  MoveL 3384 to (-30.78, 36.52, 59.84) mm, rotated rx 180 ry 0 rz 180 deg; joints [-35.866, -23.626, 89.959, 60.959, 42.078, -53.201]
  MoveL 3385 to (-30.78, 36.52, 59.84) mm, rotated rx 180 ry 0 rz 180 deg; joints [-35.866, -23.626, 89.959, 60.959, 42.078, -53.201]
  Call Extruder(71.38542)
  MoveL 3386 to (-30.58, 36.45, 59.84) mm, rotated rx 180 ry 0 rz 180 deg; joints [-35.829, -23.61, 89.95, 60.933, 42.045, -53.186]
  MoveL 3387 to (-30.58, 36.45, 59.84) mm, rotated rx 180 ry 0 rz 180 deg; joints [-35.829, -23.61, 89.95, 60.933, 42.045, -53.186]
  Call Extruder(71.51620)
  MoveL 3388 to (-30.36, 36.38, 59.84) mm, rotated rx 180 ry 0 rz 180 deg; joints [-35.788, -23.591, 89.94, 60.905, 42.009, -53.17]
  MoveL 3389 to (-30.36, 36.38, 59.84) mm, rotated rx 180 ry 0 rz 180 deg; joints [-35.788, -23.591, 89.94, 60.905, 42.009, -53.17]
  Call Extruder(71.64643)
  MoveL 3390 to (-30.14, 36.32, 59.84) mm, rotated rx 180 ry 0 rz -180 deg; joints [-35.748, -23.573, 89.929, 60.877, 41.973, -53.153]
  MoveL 3391 to (-30.14, 36.32, 59.84) mm, rotated rx 180 ry 0 rz -180 deg; joints [-35.748, -23.573, 89.929, 60.877, 41.973, -53.153]
  Call Extruder(71.77608)
  MoveL 3392 to (-29.91, 36.25, 59.84) mm, rotated rx -180 ry 0 rz 180 deg; joints [-35.708, -23.555, 89.919, 60.848, 41.937, -53.137]
  MoveL 3393 to (-29.91, 36.25, 59.84) mm, rotated rx -180 ry 0 rz 180 deg; joints [-35.708, -23.555, 89.919, 60.848, 41.937, -53.137]
  Call Extruder(71.90518)
  MoveL 3394 to (-29.69, 36.18, 59.84) mm, rotated rx 180 ry 0 rz 180 deg; joints [-35.668, -23.536, 89.908, 60.82, 41.9, -53.121]
  MoveL 3395 to (-29.69, 36.18, 59.84) mm, rotated rx 180 ry 0 rz 180 deg; joints [-35.668, -23.536, 89.908, 60.82, 41.9, -53.121]
  Call Extruder(72.02025)
  MoveL 3396 to (-29.48, 36.14, 59.84) mm, rotated rx 180 ry 0 rz 180 deg; joints [-35.634, -23.518, 89.898, 60.797, 41.87, -53.108]
  MoveL 3397 to (-29.48, 36.14, 59.84) mm, rotated rx 180 ry 0 rz 180 deg; joints [-35.634, -23.518, 89.898, 60.797, 41.87, -53.108]
  Call Extruder(72.13487)
  MoveL 3398 to (-29.28, 36.09, 59.84) mm, rotated rx -180 ry 0 rz 180 deg; joints [-35.601, -23.5, 89.888, 60.775, 41.839, -53.096]
  MoveL 3399 to (-29.28, 36.09, 59.84) mm, rotated rx -180 ry 0 rz 180 deg; joints [-35.601, -23.5, 89.888, 60.775, 41.839, -53.096]
  Call Extruder(72.24904)
  MoveL 3400 to (-29.08, 36.05, 59.84) mm, rotated rx -180 ry 0 rz 180 deg; joints [-35.567, -23.482, 89.878, 60.752, 41.808, -53.084]
  MoveL 3401 to (-29.08, 36.05, 59.84) mm, rotated rx -180 ry 0 rz 180 deg; joints [-35.567, -23.482, 89.878, 60.752, 41.808, -53.084]
  Call Extruder(72.36276)
  MoveL 3402 to (-28.87, 36, 59.84) mm, rotated rx 180 ry 0 rz 180 deg; joints [-35.533, -23.463, 89.867, 60.73, 41.777, -53.072]
  MoveL 3403 to (-28.87, 36, 59.84) mm, rotated rx 180 ry 0 rz 180 deg; joints [-35.533, -23.463, 89.867, 60.73, 41.777, -53.072]
  Call Extruder(72.48818)
  MoveL 3404 to (-28.64, 35.96, 59.84) mm, rotated rx 180 ry 0 rz 180 deg; joints [-35.497, -23.443, 89.856, 60.705, 41.744, -53.059]
  MoveL 3405 to (-28.64, 35.96, 59.84) mm, rotated rx 180 ry 0 rz 180 deg; joints [-35.497, -23.443, 89.856, 60.705, 41.744, -53.059]
  Call Extruder(72.62516)
  MoveL 3406 to (-28.4, 35.91, 59.84) mm, rotated rx 180 ry 0 rz 180 deg; joints [-35.457, -23.42, 89.843, 60.679, 41.707, -53.045]
  MoveL 3407 to (-28.4, 35.91, 59.84) mm, rotated rx 180 ry 0 rz 180 deg; joints [-35.457, -23.42, 89.843, 60.679, 41.707, -53.045]
  Call Extruder(72.76152)
  MoveL 3408 to (-28.15, 35.86, 59.84) mm, rotated rx 180 ry 0 rz 180 deg; joints [-35.417, -23.398, 89.83, 60.652, 41.67, -53.03]
  MoveL 3409 to (-28.15, 35.86, 59.84) mm, rotated rx 180 ry 0 rz 180 deg; joints [-35.417, -23.398, 89.83, 60.652, 41.67, -53.03]
  Call Extruder(72.89728)
  MoveL 3410 to (-27.9, 35.81, 59.84) mm, rotated rx 180 ry 0 rz 180 deg; joints [-35.377, -23.375, 89.817, 60.626, 41.634, -53.016]
  MoveL 3411 to (-27.9, 35.81, 59.84) mm, rotated rx 180 ry 0 rz 180 deg; joints [-35.377, -23.375, 89.817, 60.626, 41.634, -53.016]
  Call Extruder(73.03243)
  MoveL 3412 to (-27.65, 35.76, 59.84) mm, rotated rx 180 ry 0 rz 180 deg; joints [-35.337, -23.352, 89.804, 60.599, 41.597, -53.002]
  MoveL 3413 to (-27.65, 35.76, 59.84) mm, rotated rx 180 ry 0 rz 180 deg; joints [-35.337, -23.352, 89.804, 60.599, 41.597, -53.002]
  Call Extruder(73.16696)
  MoveL 3414 to (-27.4, 35.71, 59.84) mm, rotated rx 180 ry 0 rz 180 deg; joints [-35.297, -23.33, 89.791, 60.573, 41.56, -52.988]
  MoveL 3415 to (-27.4, 35.71, 59.84) mm, rotated rx 180 ry 0 rz 180 deg; joints [-35.297, -23.33, 89.791, 60.573, 41.56, -52.988]
  Call Extruder(73.30089)
  MoveL 3416 to (-27.15, 35.66, 59.84) mm, rotated rx 180 ry 0 rz 180 deg; joints [-35.258, -23.307, 89.778, 60.547, 41.524, -52.974]
  MoveL 3417 to (-27.15, 35.66, 59.84) mm, rotated rx 180 ry 0 rz 180 deg; joints [-35.258, -23.307, 89.778, 60.547, 41.524, -52.974]
  Call Extruder(73.44875)
  MoveL 3418 to (-26.87, 35.61, 59.84) mm, rotated rx 180 ry 0 rz -180 deg; joints [-35.215, -23.281, 89.764, 60.518, 41.484, -52.959]
  MoveL 3419 to (-26.87, 35.61, 59.84) mm, rotated rx 180 ry 0 rz -180 deg; joints [-35.215, -23.281, 89.764, 60.518, 41.484, -52.959]
  Call Extruder(73.61048)
  MoveL 3420 to (-26.57, 35.56, 59.84) mm, rotated rx 180 ry 0 rz 180 deg; joints [-35.168, -23.252, 89.747, 60.488, 41.441, -52.944]
  MoveL 3421 to (-26.57, 35.56, 59.84) mm, rotated rx 180 ry 0 rz 180 deg; joints [-35.168, -23.252, 89.747, 60.488, 41.441, -52.944]
  Call Extruder(73.77149)
  MoveL 3422 to (-26.26, 35.51, 59.84) mm, rotated rx 180 ry 0 rz 180 deg; joints [-35.122, -23.223, 89.731, 60.458, 41.398, -52.929]
  MoveL 3423 to (-26.26, 35.51, 59.84) mm, rotated rx 180 ry 0 rz 180 deg; joints [-35.122, -23.223, 89.731, 60.458, 41.398, -52.929]
  Call Extruder(73.93177)
  MoveL 3424 to (-25.96, 35.47, 59.84) mm, rotated rx 180 ry 0 rz 180 deg; joints [-35.075, -23.194, 89.714, 60.428, 41.355, -52.913]
  MoveL 3425 to (-25.96, 35.47, 59.84) mm, rotated rx 180 ry 0 rz 180 deg; joints [-35.075, -23.194, 89.714, 60.428, 41.355, -52.913]
  Call Extruder(74.09132)
  MoveL 3426 to (-25.65, 35.42, 59.84) mm, rotated rx 180 ry 0 rz 180 deg; joints [-35.029, -23.165, 89.698, 60.398, 41.312, -52.898]
  MoveL 3427 to (-25.65, 35.42, 59.84) mm, rotated rx 180 ry 0 rz 180 deg; joints [-35.029, -23.165, 89.698, 60.398, 41.312, -52.898]
  Call Extruder(74.25014)
  MoveL 3428 to (-25.34, 35.37, 59.84) mm, rotated rx 180 ry 0 rz 180 deg; joints [-34.983, -23.136, 89.681, 60.368, 41.269, -52.882]
  MoveL 3429 to (-25.34, 35.37, 59.84) mm, rotated rx 180 ry 0 rz 180 deg; joints [-34.983, -23.136, 89.681, 60.368, 41.269, -52.882]
  Call Extruder(74.42881)
  MoveL 3430 to (-25, 35.32, 59.84) mm, rotated rx -180 ry 0 rz -180 deg; joints [-34.932, -23.103, 89.662, 60.336, 41.221, -52.866]
  MoveL 3431 to (-25, 35.32, 59.84) mm, rotated rx -180 ry 0 rz -180 deg; joints [-34.932, -23.103, 89.662, 60.336, 41.221, -52.866]
  Call Extruder(74.62725)
  MoveL 3432 to (-24.61, 35.28, 59.84) mm, rotated rx -180 ry 0 rz 180 deg; joints [-34.877, -23.065, 89.64, 60.301, 41.169, -52.849]
  MoveL 3433 to (-24.61, 35.28, 59.84) mm, rotated rx -180 ry 0 rz 180 deg; joints [-34.877, -23.065, 89.64, 60.301, 41.169, -52.849]
  Call Extruder(74.82483)
  MoveL 3434 to (-24.22, 35.23, 59.84) mm, rotated rx 180 ry 0 rz -180 deg; joints [-34.821, -23.027, 89.618, 60.266, 41.117, -52.832]
  MoveL 3435 to (-24.22, 35.23, 59.84) mm, rotated rx 180 ry 0 rz -180 deg; joints [-34.821, -23.027, 89.618, 60.266, 41.117, -52.832]
  Call Extruder(75.02153)
  MoveL 3436 to (-23.84, 35.18, 59.84) mm, rotated rx 180 ry 0 rz -180 deg; joints [-34.766, -22.989, 89.596, 60.232, 41.065, -52.815]
  MoveL 3437 to (-23.84, 35.18, 59.84) mm, rotated rx 180 ry 0 rz -180 deg; joints [-34.766, -22.989, 89.596, 60.232, 41.065, -52.815]
  Call Extruder(75.21737)
  MoveL 3438 to (-23.45, 35.14, 59.84) mm, rotated rx -180 ry 0 rz -180 deg; joints [-34.711, -22.951, 89.574, 60.197, 41.013, -52.799]
  MoveL 3439 to (-23.45, 35.14, 59.84) mm, rotated rx -180 ry 0 rz -180 deg; joints [-34.711, -22.951, 89.574, 60.197, 41.013, -52.799]
  Call Extruder(75.51277)
  MoveL 3440 to (-22.86, 35.09, 59.84) mm, rotated rx 180 ry 0 rz 180 deg; joints [-34.631, -22.891, 89.54, 60.149, 40.937, -52.777]
  MoveL 3441 to (-22.86, 35.09, 59.84) mm, rotated rx 180 ry 0 rz 180 deg; joints [-34.631, -22.891, 89.54, 60.149, 40.937, -52.777]
  Call Extruder(75.80683)
  MoveL 3442 to (-22.27, 35.05, 59.84) mm, rotated rx 180 ry 0 rz -180 deg; joints [-34.552, -22.831, 89.505, 60.101, 40.861, -52.755]
  MoveL 3443 to (-22.27, 35.05, 59.84) mm, rotated rx 180 ry 0 rz -180 deg; joints [-34.552, -22.831, 89.505, 60.101, 40.861, -52.755]
  Call Extruder(76.09956)
  MoveL 3444 to (-21.68, 35, 59.84) mm, rotated rx 180 ry 0 rz -180 deg; joints [-34.473, -22.771, 89.47, 60.053, 40.786, -52.733]
  MoveL 3445 to (-21.68, 35, 59.84) mm, rotated rx 180 ry 0 rz -180 deg; joints [-34.473, -22.771, 89.47, 60.053, 40.786, -52.733]
  Call Extruder(76.67301)
  MoveL 3446 to (-20.52, 34.95, 59.84) mm, rotated rx 180 ry 0 rz 180 deg; joints [-34.326, -22.649, 89.399, 59.968, 40.643, -52.697]
  MoveL 3447 to (-20.52, 34.95, 59.84) mm, rotated rx 180 ry 0 rz 180 deg; joints [-34.326, -22.649, 89.399, 59.968, 40.643, -52.697]
  Call Extruder(77.38698)
  MoveL 3448 to (-19.06, 34.91, 59.84) mm, rotated rx 180 ry 0 rz 180 deg; joints [-34.146, -22.494, 89.309, 59.865, 40.468, -52.655]
  Call Extruder(194.23372)
  MoveL 3449 to (219.06, 34.91, 59.84) mm, rotated rx -180 ry 0 rz 180 deg; joints [-18.248, 9.606, 60.976, 44.762, 26.403, -41.614]
  Call Extruder(194.66228)
  MoveL 3450 to (219.94, 34.93, 59.84) mm, rotated rx 180 ry 0 rz 180 deg; joints [-18.218, 9.755, 60.801, 44.675, 26.402, -41.528]
  MoveL 3451 to (219.94, 34.93, 59.84) mm, rotated rx 180 ry 0 rz 180 deg; joints [-18.218, 9.755, 60.801, 44.675, 26.402, -41.528]
  Call Extruder(195.23572)
  MoveL 3452 to (221.1, 34.98, 59.84) mm, rotated rx 180 ry 0 rz 180 deg; joints [-18.181, 9.955, 60.565, 44.562, 26.402, -41.415]
  MoveL 3453 to (221.1, 34.98, 59.84) mm, rotated rx 180 ry 0 rz 180 deg; joints [-18.181, 9.955, 60.565, 44.562, 26.402, -41.415]
  Call Extruder(195.67004)
  MoveL 3454 to (221.97, 35.02, 59.84) mm, rotated rx 180 ry 0 rz 180 deg; joints [-18.154, 10.106, 60.386, 44.478, 26.404, -41.331]
  MoveL 3455 to (221.97, 35.02, 59.84) mm, rotated rx 180 ry 0 rz 180 deg; joints [-18.154, 10.106, 60.386, 44.478, 26.404, -41.331]
  Call Extruder(195.96409)
  MoveL 3456 to (222.56, 35.07, 59.84) mm, rotated rx 180 ry 0 rz 180 deg; joints [-18.138, 10.21, 60.264, 44.424, 26.407, -41.277]
  MoveL 3457 to (222.56, 35.07, 59.84) mm, rotated rx 180 ry 0 rz 180 deg; joints [-18.138, 10.21, 60.264, 44.424, 26.407, -41.277]
  Call Extruder(196.25948)
  MoveL 3458 to (223.15, 35.11, 59.84) mm, rotated rx -180 ry 0 rz 180 deg; joints [-18.121, 10.313, 60.142, 44.369, 26.41, -41.222]
  MoveL 3459 to (223.15, 35.11, 59.84) mm, rotated rx -180 ry 0 rz 180 deg; joints [-18.121, 10.313, 60.142, 44.369, 26.41, -41.222]
  Call Extruder(196.50572)
  MoveL 3460 to (223.64, 35.16, 59.84) mm, rotated rx 180 ry 0 rz 180 deg; joints [-18.109, 10.399, 60.039, 44.325, 26.413, -41.178]
  MoveL 3461 to (223.64, 35.16, 59.84) mm, rotated rx 180 ry 0 rz 180 deg; joints [-18.109, 10.399, 60.039, 44.325, 26.413, -41.178]
  Call Extruder(196.70242)
  MoveL 3462 to (224.03, 35.21, 59.84) mm, rotated rx 180 ry 0 rz -180 deg; joints [-18.1, 10.468, 59.957, 44.292, 26.417, -41.144]
  MoveL 3463 to (224.03, 35.21, 59.84) mm, rotated rx 180 ry 0 rz -180 deg; joints [-18.1, 10.468, 59.957, 44.292, 26.417, -41.144]
  Call Extruder(196.90000)
  MoveL 3464 to (224.42, 35.25, 59.84) mm, rotated rx -180 ry 0 rz 180 deg; joints [-18.091, 10.537, 59.875, 44.258, 26.42, -41.11]
  MoveL 3465 to (224.42, 35.25, 59.84) mm, rotated rx -180 ry 0 rz 180 deg; joints [-18.091, 10.537, 59.875, 44.258, 26.42, -41.11]
  Call Extruder(197.09844)
  MoveL 3466 to (224.8, 35.3, 59.84) mm, rotated rx 180 ry 0 rz 180 deg; joints [-18.082, 10.607, 59.793, 44.225, 26.424, -41.076]
  MoveL 3467 to (224.8, 35.3, 59.84) mm, rotated rx 180 ry 0 rz 180 deg; joints [-18.082, 10.607, 59.793, 44.225, 26.424, -41.076]
  Call Extruder(197.29775)
  MoveL 3468 to (225.19, 35.34, 59.84) mm, rotated rx 180 ry 0 rz 180 deg; joints [-18.073, 10.676, 59.71, 44.191, 26.427, -41.042]
  MoveL 3469 to (225.19, 35.34, 59.84) mm, rotated rx 180 ry 0 rz 180 deg; joints [-18.073, 10.676, 59.71, 44.191, 26.427, -41.042]
  Call Extruder(197.45657)
  MoveL 3470 to (225.5, 35.39, 59.84) mm, rotated rx 180 ry 0 rz -180 deg; joints [-18.068, 10.731, 59.644, 44.166, 26.431, -41.016]
  MoveL 3471 to (225.5, 35.39, 59.84) mm, rotated rx 180 ry 0 rz -180 deg; joints [-18.068, 10.731, 59.644, 44.166, 26.431, -41.016]
  Call Extruder(197.61612)
  MoveL 3472 to (225.8, 35.44, 59.84) mm, rotated rx 180 ry 0 rz 180 deg; joints [-18.062, 10.787, 59.578, 44.142, 26.435, -40.991]
  MoveL 3473 to (225.8, 35.44, 59.84) mm, rotated rx 180 ry 0 rz 180 deg; joints [-18.062, 10.787, 59.578, 44.142, 26.435, -40.991]
  Call Extruder(197.77640)
  MoveL 3474 to (226.11, 35.49, 59.84) mm, rotated rx 180 ry 0 rz 180 deg; joints [-18.056, 10.842, 59.511, 44.117, 26.439, -40.965]
  MoveL 3475 to (226.11, 35.49, 59.84) mm, rotated rx 180 ry 0 rz 180 deg; joints [-18.056, 10.842, 59.511, 44.117, 26.439, -40.965]
  Call Extruder(197.93740)
  MoveL 3476 to (226.41, 35.54, 59.84) mm, rotated rx 180 ry 0 rz -180 deg; joints [-18.051, 10.898, 59.445, 44.092, 26.444, -40.94]
  MoveL 3477 to (226.41, 35.54, 59.84) mm, rotated rx 180 ry 0 rz -180 deg; joints [-18.051, 10.898, 59.445, 44.092, 26.444, -40.94]
  Call Extruder(198.09914)
  MoveL 3478 to (226.72, 35.59, 59.84) mm, rotated rx -180 ry 0 rz 180 deg; joints [-18.045, 10.954, 59.378, 44.067, 26.448, -40.914]
  MoveL 3479 to (226.72, 35.59, 59.84) mm, rotated rx -180 ry 0 rz 180 deg; joints [-18.045, 10.954, 59.378, 44.067, 26.448, -40.914]
  Call Extruder(198.26160)
  MoveL 3480 to (227.03, 35.64, 59.84) mm, rotated rx 180 ry 0 rz 180 deg; joints [-18.039, 11.009, 59.312, 44.043, 26.452, -40.888]
  MoveL 3481 to (227.03, 35.64, 59.84) mm, rotated rx 180 ry 0 rz 180 deg; joints [-18.039, 11.009, 59.312, 44.043, 26.452, -40.888]
  Call Extruder(198.39552)
  MoveL 3482 to (227.28, 35.68, 59.84) mm, rotated rx -180 ry 0 rz 180 deg; joints [-18.036, 11.055, 59.256, 44.024, 26.456, -40.869]
  MoveL 3483 to (227.28, 35.68, 59.84) mm, rotated rx -180 ry 0 rz 180 deg; joints [-18.036, 11.055, 59.256, 44.024, 26.456, -40.869]
  Call Extruder(198.53006)
  MoveL 3484 to (227.52, 35.73, 59.84) mm, rotated rx 180 ry 0 rz -180 deg; joints [-18.033, 11.101, 59.201, 44.005, 26.461, -40.849]
  MoveL 3485 to (227.52, 35.73, 59.84) mm, rotated rx 180 ry 0 rz -180 deg; joints [-18.033, 11.101, 59.201, 44.005, 26.461, -40.849]
  Call Extruder(198.66521)
  MoveL 3486 to (227.77, 35.78, 59.84) mm, rotated rx 180 ry 0 rz 180 deg; joints [-18.029, 11.147, 59.146, 43.986, 26.465, -40.83]
  MoveL 3487 to (227.77, 35.78, 59.84) mm, rotated rx 180 ry 0 rz 180 deg; joints [-18.029, 11.147, 59.146, 43.986, 26.465, -40.83]
  Call Extruder(198.80097)
  MoveL 3488 to (228.02, 35.83, 59.84) mm, rotated rx -180 ry 0 rz 180 deg; joints [-18.026, 11.193, 59.091, 43.967, 26.469, -40.81]
  MoveL 3489 to (228.02, 35.83, 59.84) mm, rotated rx -180 ry 0 rz 180 deg; joints [-18.026, 11.193, 59.091, 43.967, 26.469, -40.81]
  Call Extruder(198.93734)
  MoveL 3490 to (228.27, 35.88, 59.84) mm, rotated rx 180 ry 0 rz 180 deg; joints [-18.022, 11.24, 59.035, 43.949, 26.474, -40.79]
  MoveL 3491 to (228.27, 35.88, 59.84) mm, rotated rx 180 ry 0 rz 180 deg; joints [-18.022, 11.24, 59.035, 43.949, 26.474, -40.79]
  Call Extruder(199.07431)
  MoveL 3492 to (228.52, 35.93, 59.84) mm, rotated rx -180 ry 0 rz 180 deg; joints [-18.019, 11.286, 58.98, 43.93, 26.478, -40.77]
  MoveL 3493 to (228.52, 35.93, 59.84) mm, rotated rx -180 ry 0 rz 180 deg; joints [-18.019, 11.286, 58.98, 43.93, 26.478, -40.77]
  Call Extruder(199.21190)
  MoveL 3494 to (228.77, 35.98, 59.84) mm, rotated rx 180 ry 0 rz 180 deg; joints [-18.015, 11.332, 58.924, 43.911, 26.483, -40.75]
  MoveL 3495 to (228.77, 35.98, 59.84) mm, rotated rx 180 ry 0 rz 180 deg; joints [-18.015, 11.332, 58.924, 43.911, 26.483, -40.75]
  Call Extruder(199.32562)
  MoveL 3496 to (228.97, 36.03, 59.84) mm, rotated rx 180 ry 0 rz 180 deg; joints [-18.013, 11.37, 58.878, 43.896, 26.487, -40.734]
  MoveL 3497 to (228.97, 36.03, 59.84) mm, rotated rx 180 ry 0 rz 180 deg; joints [-18.013, 11.37, 58.878, 43.896, 26.487, -40.734]
  Call Extruder(199.43979)
  MoveL 3498 to (229.18, 36.07, 59.84) mm, rotated rx 180 ry 0 rz 180 deg; joints [-18.01, 11.408, 58.832, 43.881, 26.491, -40.719]
  MoveL 3499 to (229.18, 36.07, 59.84) mm, rotated rx 180 ry 0 rz 180 deg; joints [-18.01, 11.408, 58.832, 43.881, 26.491, -40.719]
  Call Extruder(199.55441)
  MoveL 3500 to (229.38, 36.12, 59.84) mm, rotated rx -180 ry 0 rz -180 deg; joints [-18.008, 11.446, 58.786, 43.866, 26.495, -40.703]
  MoveL 3501 to (229.38, 36.12, 59.84) mm, rotated rx -180 ry 0 rz -180 deg; joints [-18.008, 11.446, 58.786, 43.866, 26.495, -40.703]
  Call Extruder(199.66948)
  MoveL 3502 to (229.59, 36.16, 59.84) mm, rotated rx 180 ry 0 rz 180 deg; joints [-18.006, 11.485, 58.74, 43.851, 26.499, -40.687]
  MoveL 3503 to (229.59, 36.16, 59.84) mm, rotated rx 180 ry 0 rz 180 deg; joints [-18.006, 11.485, 58.74, 43.851, 26.499, -40.687]
  Call Extruder(199.79172)
  MoveL 3504 to (229.8, 36.22, 59.84) mm, rotated rx -180 ry 0 rz 180 deg; joints [-18.004, 11.525, 58.691, 43.837, 26.505, -40.672]
  MoveL 3505 to (229.8, 36.22, 59.84) mm, rotated rx -180 ry 0 rz 180 deg; joints [-18.004, 11.525, 58.691, 43.837, 26.505, -40.672]
  Call Extruder(199.92138)
  MoveL 3506 to (230.02, 36.28, 59.84) mm, rotated rx 180 ry 0 rz 180 deg; joints [-18.004, 11.568, 58.639, 43.823, 26.511, -40.657]
  MoveL 3507 to (230.02, 36.28, 59.84) mm, rotated rx 180 ry 0 rz 180 deg; joints [-18.004, 11.568, 58.639, 43.823, 26.511, -40.657]
  Call Extruder(200.05161)
  MoveL 3508 to (230.25, 36.35, 59.84) mm, rotated rx 180 ry 0 rz 180 deg; joints [-18.003, 11.611, 58.587, 43.81, 26.517, -40.642]
  MoveL 3509 to (230.25, 36.35, 59.84) mm, rotated rx 180 ry 0 rz 180 deg; joints [-18.003, 11.611, 58.587, 43.81, 26.517, -40.642]
  Call Extruder(200.18241)
  MoveL 3510 to (230.47, 36.42, 59.84) mm, rotated rx 180 ry 0 rz -180 deg; joints [-18.003, 11.654, 58.535, 43.796, 26.523, -40.627]
  MoveL 3511 to (230.47, 36.42, 59.84) mm, rotated rx 180 ry 0 rz -180 deg; joints [-18.003, 11.654, 58.535, 43.796, 26.523, -40.627]
  Call Extruder(200.31377)
  MoveL 3512 to (230.69, 36.49, 59.84) mm, rotated rx -180 ry 0 rz -180 deg; joints [-18.002, 11.697, 58.482, 43.783, 26.529, -40.612]
  MoveL 3513 to (230.69, 36.49, 59.84) mm, rotated rx -180 ry 0 rz -180 deg; joints [-18.002, 11.697, 58.482, 43.783, 26.529, -40.612]
  Call Extruder(200.43194)
  MoveL 3514 to (230.89, 36.55, 59.84) mm, rotated rx -180 ry 0 rz 180 deg; joints [-18.002, 11.736, 58.436, 43.772, 26.535, -40.6]
  MoveL 3515 to (230.89, 36.55, 59.84) mm, rotated rx -180 ry 0 rz 180 deg; joints [-18.002, 11.736, 58.436, 43.772, 26.535, -40.6]
  Call Extruder(200.55059)
  MoveL 3516 to (231.09, 36.62, 59.84) mm, rotated rx -180 ry 0 rz 180 deg; joints [-18.002, 11.775, 58.389, 43.76, 26.541, -40.587]
  MoveL 3517 to (231.09, 36.62, 59.84) mm, rotated rx -180 ry 0 rz 180 deg; joints [-18.002, 11.775, 58.389, 43.76, 26.541, -40.587]
  Call Extruder(200.66975)
  MoveL 3518 to (231.29, 36.68, 59.84) mm, rotated rx 180 ry 0 rz 180 deg; joints [-18.002, 11.813, 58.342, 43.749, 26.547, -40.574]
  MoveL 3519 to (231.29, 36.68, 59.84) mm, rotated rx 180 ry 0 rz 180 deg; joints [-18.002, 11.813, 58.342, 43.749, 26.547, -40.574]
  Call Extruder(200.77883)
  MoveL 3520 to (231.47, 36.74, 59.84) mm, rotated rx -180 ry 0 rz 180 deg; joints [-18.002, 11.849, 58.299, 43.738, 26.552, -40.563]
  MoveL 3521 to (231.47, 36.74, 59.84) mm, rotated rx -180 ry 0 rz 180 deg; joints [-18.002, 11.849, 58.299, 43.738, 26.552, -40.563]
  Call Extruder(200.87772)
  MoveL 3522 to (231.64, 36.79, 59.84) mm, rotated rx 180 ry 0 rz 180 deg; joints [-18.002, 11.88, 58.26, 43.729, 26.557, -40.552]
  MoveL 3523 to (231.64, 36.79, 59.84) mm, rotated rx 180 ry 0 rz 180 deg; joints [-18.002, 11.88, 58.26, 43.729, 26.557, -40.552]
  Call Extruder(201.05968)
  MoveL 3524 to (231.93, 36.91, 59.84) mm, rotated rx 180 ry 0 rz 180 deg; joints [-18.005, 11.939, 58.19, 43.716, 26.568, -40.537]
  MoveL 3525 to (231.93, 36.91, 59.84) mm, rotated rx 180 ry 0 rz 180 deg; joints [-18.005, 11.939, 58.19, 43.716, 26.568, -40.537]
  Call Extruder(201.24239)
  MoveL 3526 to (232.22, 37.04, 59.84) mm, rotated rx 180 ry 0 rz -180 deg; joints [-18.008, 11.997, 58.119, 43.704, 26.579, -40.522]
  MoveL 3527 to (232.22, 37.04, 59.84) mm, rotated rx 180 ry 0 rz -180 deg; joints [-18.008, 11.997, 58.119, 43.704, 26.579, -40.522]
  Call Extruder(201.41281)
  MoveL 3528 to (232.49, 37.15, 59.84) mm, rotated rx -180 ry 0 rz -180 deg; joints [-18.011, 12.051, 58.053, 43.692, 26.59, -40.508]
  MoveL 3529 to (232.49, 37.15, 59.84) mm, rotated rx -180 ry 0 rz -180 deg; joints [-18.011, 12.051, 58.053, 43.692, 26.59, -40.508]
  Call Extruder(201.57081)
  MoveL 3530 to (232.74, 37.26, 59.84) mm, rotated rx 180 ry 0 rz 180 deg; joints [-18.013, 12.102, 57.991, 43.682, 26.599, -40.495]
  MoveL 3531 to (232.74, 37.26, 59.84) mm, rotated rx 180 ry 0 rz 180 deg; joints [-18.013, 12.102, 57.991, 43.682, 26.599, -40.495]
  Call Extruder(201.72941)
  MoveL 3532 to (232.99, 37.36, 59.84) mm, rotated rx -180 ry 0 rz 180 deg; joints [-18.016, 12.152, 57.93, 43.672, 26.609, -40.483]
  MoveL 3533 to (232.99, 37.36, 59.84) mm, rotated rx -180 ry 0 rz 180 deg; joints [-18.016, 12.152, 57.93, 43.672, 26.609, -40.483]
  Call Extruder(201.93558)
  MoveL 3534 to (233.29, 37.54, 59.84) mm, rotated rx 180 ry 0 rz -180 deg; joints [-18.024, 12.216, 57.852, 43.666, 26.625, -40.473]
  MoveL 3535 to (233.29, 37.54, 59.84) mm, rotated rx 180 ry 0 rz -180 deg; joints [-18.024, 12.216, 57.852, 43.666, 26.625, -40.473]
  Call Extruder(202.14252)
  MoveL 3536 to (233.6, 37.71, 59.84) mm, rotated rx 180 ry 0 rz 180 deg; joints [-18.033, 12.28, 57.774, 43.661, 26.64, -40.464]
  MoveL 3537 to (233.6, 37.71, 59.84) mm, rotated rx 180 ry 0 rz 180 deg; joints [-18.033, 12.28, 57.774, 43.661, 26.64, -40.464]
  Call Extruder(202.35025)
  MoveL 3538 to (233.9, 37.89, 59.84) mm, rotated rx -180 ry 0 rz 180 deg; joints [-18.041, 12.344, 57.696, 43.655, 26.656, -40.455]
  MoveL 3539 to (233.9, 37.89, 59.84) mm, rotated rx -180 ry 0 rz 180 deg; joints [-18.041, 12.344, 57.696, 43.655, 26.656, -40.455]
  Call Extruder(202.55875)
  MoveL 3540 to (234.21, 38.07, 59.84) mm, rotated rx 180 ry 0 rz 180 deg; joints [-18.049, 12.408, 57.617, 43.65, 26.672, -40.445]
  MoveL 3541 to (234.21, 38.07, 59.84) mm, rotated rx 180 ry 0 rz 180 deg; joints [-18.049, 12.408, 57.617, 43.65, 26.672, -40.445]
  Call Extruder(202.73829)
  MoveL 3542 to (234.45, 38.24, 59.84) mm, rotated rx -180 ry 0 rz 180 deg; joints [-18.06, 12.462, 57.551, 43.651, 26.687, -40.443]
  MoveL 3543 to (234.45, 38.24, 59.84) mm, rotated rx -180 ry 0 rz 180 deg; joints [-18.06, 12.462, 57.551, 43.651, 26.687, -40.443]
  Call Extruder(203.07171)
  MoveL 3544 to (234.9, 38.57, 59.84) mm, rotated rx 180 ry 0 rz 180 deg; joints [-18.079, 12.561, 57.429, 43.653, 26.716, -40.438]
  MoveL 3545 to (234.9, 38.57, 59.84) mm, rotated rx 180 ry 0 rz 180 deg; joints [-18.079, 12.561, 57.429, 43.653, 26.716, -40.438]
  Call Extruder(203.40631)
  MoveL 3546 to (235.35, 38.9, 59.84) mm, rotated rx 180 ry 0 rz 180 deg; joints [-18.099, 12.661, 57.307, 43.655, 26.745, -40.432]
  Call Extruder(204.23426)
  MoveL 3547 to (236.39, 39.81, 59.84) mm, rotated rx 180 ry 0 rz -180 deg; joints [-18.16, 12.9, 57.013, 43.683, 26.825, -40.441]
  Call Extruder(205.06220)
  MoveL 3548 to (237.3, 40.85, 59.84) mm, rotated rx 180 ry 0 rz 180 deg; joints [-18.24, 13.125, 56.735, 43.745, 26.915, -40.479]
  Call Extruder(205.22950)
  MoveL 3549 to (237.47, 41.07, 59.84) mm, rotated rx 180 ry 0 rz 180 deg; joints [-18.258, 13.168, 56.682, 43.762, 26.934, -40.491]
  MoveL 3550 to (237.47, 41.07, 59.84) mm, rotated rx 180 ry 0 rz 180 deg; joints [-18.258, 13.168, 56.682, 43.762, 26.934, -40.491]
  Call Extruder(205.56292)
  MoveL 3551 to (237.79, 41.52, 59.84) mm, rotated rx -180 ry 0 rz 180 deg; joints [-18.295, 13.254, 56.575, 43.795, 26.973, -40.514]
  MoveL 3552 to (237.79, 41.52, 59.84) mm, rotated rx -180 ry 0 rz 180 deg; joints [-18.295, 13.254, 56.575, 43.795, 26.973, -40.514]
  Call Extruder(205.89514)
  MoveL 3553 to (238.12, 41.97, 59.84) mm, rotated rx -180 ry 0 rz -180 deg; joints [-18.332, 13.34, 56.468, 43.829, 27.012, -40.537]
  MoveL 3554 to (238.12, 41.97, 59.84) mm, rotated rx -180 ry 0 rz -180 deg; joints [-18.332, 13.34, 56.468, 43.829, 27.012, -40.537]
  Call Extruder(206.01284)
  MoveL 3555 to (238.22, 42.15, 59.84) mm, rotated rx 180 ry 0 rz 180 deg; joints [-18.346, 13.368, 56.433, 43.844, 27.026, -40.549]
  MoveL 3556 to (238.22, 42.15, 59.84) mm, rotated rx 180 ry 0 rz 180 deg; joints [-18.346, 13.368, 56.433, 43.844, 27.026, -40.549]
  Call Extruder(206.22057)
  MoveL 3557 to (238.4, 42.45, 59.84) mm, rotated rx 180 ry 0 rz 180 deg; joints [-18.373, 13.419, 56.371, 43.872, 27.052, -40.57]
  MoveL 3558 to (238.4, 42.45, 59.84) mm, rotated rx 180 ry 0 rz 180 deg; joints [-18.373, 13.419, 56.371, 43.872, 27.052, -40.57]
  Call Extruder(206.42751)
  MoveL 3559 to (238.57, 42.75, 59.84) mm, rotated rx 180 ry 0 rz 180 deg; joints [-18.399, 13.468, 56.309, 43.899, 27.078, -40.59]
  MoveL 3560 to (238.57, 42.75, 59.84) mm, rotated rx 180 ry 0 rz 180 deg; joints [-18.399, 13.468, 56.309, 43.899, 27.078, -40.59]
  Call Extruder(206.63368)
  MoveL 3561 to (238.75, 43.06, 59.84) mm, rotated rx -180 ry 0 rz 180 deg; joints [-18.425, 13.519, 56.246, 43.926, 27.104, -40.611]
  MoveL 3562 to (238.75, 43.06, 59.84) mm, rotated rx -180 ry 0 rz 180 deg; joints [-18.425, 13.519, 56.246, 43.926, 27.104, -40.611]
  Call Extruder(206.81537)
  MoveL 3563 to (238.89, 43.34, 59.84) mm, rotated rx 180 ry 0 rz -180 deg; joints [-18.45, 13.561, 56.194, 43.953, 27.127, -40.631]
  MoveL 3564 to (238.89, 43.34, 59.84) mm, rotated rx 180 ry 0 rz -180 deg; joints [-18.45, 13.561, 56.194, 43.953, 27.127, -40.631]
  Call Extruder(206.97338)
  MoveL 3565 to (239, 43.58, 59.84) mm, rotated rx -180 ry 0 rz 180 deg; joints [-18.472, 13.595, 56.151, 43.979, 27.148, -40.652]
  MoveL 3566 to (239, 43.58, 59.84) mm, rotated rx -180 ry 0 rz 180 deg; joints [-18.472, 13.595, 56.151, 43.979, 27.148, -40.652]
  Call Extruder(207.13078)
  MoveL 3567 to (239.11, 43.83, 59.84) mm, rotated rx 180 ry 0 rz 180 deg; joints [-18.495, 13.63, 56.108, 44.005, 27.169, -40.672]
  MoveL 3568 to (239.11, 43.83, 59.84) mm, rotated rx 180 ry 0 rz 180 deg; joints [-18.495, 13.63, 56.108, 44.005, 27.169, -40.672]
  Call Extruder(207.31350)
  MoveL 3569 to (239.23, 44.13, 59.84) mm, rotated rx 180 ry 0 rz 180 deg; joints [-18.522, 13.67, 56.058, 44.037, 27.194, -40.697]
  MoveL 3570 to (239.23, 44.13, 59.84) mm, rotated rx 180 ry 0 rz 180 deg; joints [-18.522, 13.67, 56.058, 44.037, 27.194, -40.697]
  Call Extruder(207.49546)
  MoveL 3571 to (239.35, 44.42, 59.84) mm, rotated rx -180 ry 0 rz 180 deg; joints [-18.549, 13.709, 56.009, 44.068, 27.218, -40.722]
  MoveL 3572 to (239.35, 44.42, 59.84) mm, rotated rx -180 ry 0 rz 180 deg; joints [-18.549, 13.709, 56.009, 44.068, 27.218, -40.722]
  Call Extruder(207.64279)
  MoveL 3573 to (239.44, 44.66, 59.84) mm, rotated rx 180 ry 0 rz 180 deg; joints [-18.571, 13.741, 55.97, 44.094, 27.238, -40.743]
  MoveL 3574 to (239.44, 44.66, 59.84) mm, rotated rx 180 ry 0 rz 180 deg; joints [-18.571, 13.741, 55.97, 44.094, 27.238, -40.743]
  Call Extruder(207.75602)
  MoveL 3575 to (239.5, 44.85, 59.84) mm, rotated rx 180 ry 0 rz 180 deg; joints [-18.589, 13.763, 55.941, 44.116, 27.254, -40.76]
  MoveL 3576 to (239.5, 44.85, 59.84) mm, rotated rx 180 ry 0 rz 180 deg; joints [-18.589, 13.763, 55.941, 44.116, 27.254, -40.76]
  Call Extruder(207.86881)
  MoveL 3577 to (239.56, 45.03, 59.84) mm, rotated rx 180 ry 0 rz 180 deg; joints [-18.607, 13.786, 55.913, 44.138, 27.27, -40.778]
  MoveL 3578 to (239.56, 45.03, 59.84) mm, rotated rx 180 ry 0 rz 180 deg; joints [-18.607, 13.786, 55.913, 44.138, 27.27, -40.778]
  Call Extruder(207.98116)
  MoveL 3579 to (239.62, 45.22, 59.84) mm, rotated rx -180 ry 0 rz 180 deg; joints [-18.625, 13.809, 55.885, 44.16, 27.285, -40.796]
  MoveL 3580 to (239.62, 45.22, 59.84) mm, rotated rx -180 ry 0 rz 180 deg; joints [-18.625, 13.809, 55.885, 44.16, 27.285, -40.796]
  Call Extruder(208.09306)
  MoveL 3581 to (239.68, 45.41, 59.84) mm, rotated rx 180 ry 0 rz 180 deg; joints [-18.642, 13.831, 55.856, 44.182, 27.301, -40.813]
  MoveL 3582 to (239.68, 45.41, 59.84) mm, rotated rx 180 ry 0 rz 180 deg; joints [-18.642, 13.831, 55.856, 44.182, 27.301, -40.813]
  Call Extruder(208.21446)
  MoveL 3583 to (239.75, 45.62, 59.84) mm, rotated rx -180 ry 0 rz 180 deg; joints [-18.662, 13.856, 55.826, 44.206, 27.318, -40.833]
  MoveL 3584 to (239.75, 45.62, 59.84) mm, rotated rx -180 ry 0 rz 180 deg; joints [-18.662, 13.856, 55.826, 44.206, 27.318, -40.833]
  Call Extruder(208.34525)
  MoveL 3585 to (239.82, 45.84, 59.84) mm, rotated rx 180 ry 0 rz 180 deg; joints [-18.683, 13.882, 55.793, 44.232, 27.337, -40.854]
  MoveL 3586 to (239.82, 45.84, 59.84) mm, rotated rx 180 ry 0 rz 180 deg; joints [-18.683, 13.882, 55.793, 44.232, 27.337, -40.854]
  Call Extruder(208.47548)
  MoveL 3587 to (239.88, 46.06, 59.84) mm, rotated rx 180 ry 0 rz 180 deg; joints [-18.705, 13.908, 55.76, 44.258, 27.356, -40.875]
  MoveL 3588 to (239.88, 46.06, 59.84) mm, rotated rx 180 ry 0 rz 180 deg; joints [-18.705, 13.908, 55.76, 44.258, 27.356, -40.875]
  Call Extruder(208.60514)
  MoveL 3589 to (239.95, 46.29, 59.84) mm, rotated rx 180 ry 0 rz 180 deg; joints [-18.726, 13.934, 55.727, 44.284, 27.374, -40.896]
  MoveL 3590 to (239.95, 46.29, 59.84) mm, rotated rx 180 ry 0 rz 180 deg; joints [-18.726, 13.934, 55.727, 44.284, 27.374, -40.896]
  Call Extruder(208.73424)
  MoveL 3591 to (240.02, 46.51, 59.84) mm, rotated rx 180 ry 0 rz 180 deg; joints [-18.747, 13.96, 55.695, 44.311, 27.393, -40.917]
  MoveL 3592 to (240.02, 46.51, 59.84) mm, rotated rx 180 ry 0 rz 180 deg; joints [-18.747, 13.96, 55.695, 44.311, 27.393, -40.917]
  Call Extruder(208.84929)
  MoveL 3593 to (240.06, 46.72, 59.84) mm, rotated rx 180 ry 0 rz 180 deg; joints [-18.767, 13.981, 55.669, 44.336, 27.41, -40.939]
  MoveL 3594 to (240.06, 46.72, 59.84) mm, rotated rx 180 ry 0 rz 180 deg; joints [-18.767, 13.981, 55.669, 44.336, 27.41, -40.939]
  Call Extruder(208.96389)
  MoveL 3595 to (240.11, 46.92, 59.84) mm, rotated rx -180 ry 0 rz 180 deg; joints [-18.787, 14.002, 55.643, 44.362, 27.427, -40.96]
  MoveL 3596 to (240.11, 46.92, 59.84) mm, rotated rx -180 ry 0 rz 180 deg; joints [-18.787, 14.002, 55.643, 44.362, 27.427, -40.96]
  Call Extruder(209.07804)
  MoveL 3597 to (240.15, 47.12, 59.84) mm, rotated rx 180 ry 0 rz 180 deg; joints [-18.807, 14.023, 55.617, 44.388, 27.444, -40.981]
  MoveL 3598 to (240.15, 47.12, 59.84) mm, rotated rx 180 ry 0 rz 180 deg; joints [-18.807, 14.023, 55.617, 44.388, 27.444, -40.981]
  Call Extruder(209.19174)
  MoveL 3599 to (240.2, 47.33, 59.84) mm, rotated rx 180 ry 0 rz 180 deg; joints [-18.827, 14.044, 55.59, 44.413, 27.461, -41.002]
  MoveL 3600 to (240.2, 47.33, 59.84) mm, rotated rx 180 ry 0 rz 180 deg; joints [-18.827, 14.044, 55.59, 44.413, 27.461, -41.002]
  Call Extruder(209.31715)
  MoveL 3601 to (240.24, 47.56, 59.84) mm, rotated rx 180 ry 0 rz 180 deg; joints [-18.85, 14.066, 55.562, 44.442, 27.479, -41.025]
  MoveL 3602 to (240.24, 47.56, 59.84) mm, rotated rx 180 ry 0 rz 180 deg; joints [-18.85, 14.066, 55.562, 44.442, 27.479, -41.025]
  Call Extruder(209.45413)
  MoveL 3603 to (240.29, 47.8, 59.84) mm, rotated rx 180 ry 0 rz 180 deg; joints [-18.874, 14.091, 55.531, 44.474, 27.5, -41.051]
  MoveL 3604 to (240.29, 47.8, 59.84) mm, rotated rx 180 ry 0 rz 180 deg; joints [-18.874, 14.091, 55.531, 44.474, 27.5, -41.051]
  Call Extruder(209.59050)
  MoveL 3605 to (240.34, 48.05, 59.84) mm, rotated rx 180 ry 0 rz 180 deg; joints [-18.899, 14.116, 55.5, 44.505, 27.521, -41.078]
  MoveL 3606 to (240.34, 48.05, 59.84) mm, rotated rx 180 ry 0 rz 180 deg; joints [-18.899, 14.116, 55.5, 44.505, 27.521, -41.078]
  Call Extruder(209.72625)
  MoveL 3607 to (240.39, 48.3, 59.84) mm, rotated rx -180 ry 0 rz 180 deg; joints [-18.923, 14.14, 55.469, 44.537, 27.541, -41.104]
  MoveL 3608 to (240.39, 48.3, 59.84) mm, rotated rx -180 ry 0 rz 180 deg; joints [-18.923, 14.14, 55.469, 44.537, 27.541, -41.104]
  Call Extruder(209.86140)
  MoveL 3609 to (240.44, 48.55, 59.84) mm, rotated rx 180 ry 0 rz 180 deg; joints [-18.948, 14.165, 55.438, 44.569, 27.562, -41.129]
  MoveL 3610 to (240.44, 48.55, 59.84) mm, rotated rx 180 ry 0 rz 180 deg; joints [-18.948, 14.165, 55.438, 44.569, 27.562, -41.129]
  Call Extruder(209.99594)
  MoveL 3611 to (240.49, 48.8, 59.84) mm, rotated rx -180 ry 0 rz 180 deg; joints [-18.973, 14.19, 55.407, 44.6, 27.583, -41.155]
  MoveL 3612 to (240.49, 48.8, 59.84) mm, rotated rx -180 ry 0 rz 180 deg; joints [-18.973, 14.19, 55.407, 44.6, 27.583, -41.155]
  Call Extruder(210.12986)
  MoveL 3613 to (240.54, 49.05, 59.84) mm, rotated rx 180 ry 0 rz 180 deg; joints [-18.997, 14.215, 55.376, 44.631, 27.603, -41.181]
  MoveL 3614 to (240.54, 49.05, 59.84) mm, rotated rx 180 ry 0 rz 180 deg; joints [-18.997, 14.215, 55.376, 44.631, 27.603, -41.181]
  Call Extruder(210.27773)
  MoveL 3615 to (240.59, 49.33, 59.84) mm, rotated rx 180 ry 0 rz 180 deg; joints [-19.025, 14.241, 55.342, 44.667, 27.626, -41.21]
  MoveL 3616 to (240.59, 49.33, 59.84) mm, rotated rx 180 ry 0 rz 180 deg; joints [-19.025, 14.241, 55.342, 44.667, 27.626, -41.21]
  Call Extruder(210.43947)
  MoveL 3617 to (240.64, 49.63, 59.84) mm, rotated rx -180 ry 0 rz 180 deg; joints [-19.055, 14.269, 55.307, 44.706, 27.652, -41.243]
  MoveL 3618 to (240.64, 49.63, 59.84) mm, rotated rx -180 ry 0 rz 180 deg; joints [-19.055, 14.269, 55.307, 44.706, 27.652, -41.243]
  Call Extruder(210.60049)
  MoveL 3619 to (240.69, 49.94, 59.84) mm, rotated rx -180 ry 0 rz 180 deg; joints [-19.086, 14.298, 55.271, 44.746, 27.677, -41.275]
  MoveL 3620 to (240.69, 49.94, 59.84) mm, rotated rx -180 ry 0 rz 180 deg; joints [-19.086, 14.298, 55.271, 44.746, 27.677, -41.275]
  Call Extruder(210.76078)
  MoveL 3621 to (240.73, 50.24, 59.84) mm, rotated rx -180 ry 0 rz 180 deg; joints [-19.116, 14.326, 55.236, 44.785, 27.702, -41.308]
  MoveL 3622 to (240.73, 50.24, 59.84) mm, rotated rx -180 ry 0 rz 180 deg; joints [-19.116, 14.326, 55.236, 44.785, 27.702, -41.308]
  Call Extruder(210.92034)
  MoveL 3623 to (240.78, 50.55, 59.84) mm, rotated rx 180 ry 0 rz 180 deg; joints [-19.146, 14.354, 55.2, 44.825, 27.727, -41.34]
  MoveL 3624 to (240.78, 50.55, 59.84) mm, rotated rx 180 ry 0 rz 180 deg; joints [-19.146, 14.354, 55.2, 44.825, 27.727, -41.34]
  Call Extruder(211.07917)
  MoveL 3625 to (240.83, 50.86, 59.84) mm, rotated rx 180 ry 0 rz 180 deg; joints [-19.177, 14.383, 55.164, 44.864, 27.753, -41.373]
  MoveL 3626 to (240.83, 50.86, 59.84) mm, rotated rx 180 ry 0 rz 180 deg; joints [-19.177, 14.383, 55.164, 44.864, 27.753, -41.373]
  Call Extruder(211.25784)
  MoveL 3627 to (240.88, 51.2, 59.84) mm, rotated rx 180 ry 0 rz -180 deg; joints [-19.212, 14.413, 55.125, 44.909, 27.781, -41.41]
  MoveL 3628 to (240.88, 51.2, 59.84) mm, rotated rx 180 ry 0 rz -180 deg; joints [-19.212, 14.413, 55.125, 44.909, 27.781, -41.41]
  Call Extruder(211.45628)
  MoveL 3629 to (240.92, 51.59, 59.84) mm, rotated rx 180 ry 0 rz 180 deg; joints [-19.251, 14.447, 55.083, 44.96, 27.814, -41.452]
  MoveL 3630 to (240.92, 51.59, 59.84) mm, rotated rx 180 ry 0 rz 180 deg; joints [-19.251, 14.447, 55.083, 44.96, 27.814, -41.452]
  Call Extruder(211.65386)
  MoveL 3631 to (240.97, 51.98, 59.84) mm, rotated rx 180 ry 0 rz 180 deg; joints [-19.29, 14.48, 55.041, 45.011, 27.846, -41.494]
  MoveL 3632 to (240.97, 51.98, 59.84) mm, rotated rx 180 ry 0 rz 180 deg; joints [-19.29, 14.48, 55.041, 45.011, 27.846, -41.494]
  Call Extruder(211.85056)
  MoveL 3633 to (241.02, 52.37, 59.84) mm, rotated rx 180 ry 0 rz -180 deg; joints [-19.329, 14.514, 54.999, 45.062, 27.878, -41.537]
  MoveL 3634 to (241.02, 52.37, 59.84) mm, rotated rx 180 ry 0 rz -180 deg; joints [-19.329, 14.514, 54.999, 45.062, 27.878, -41.537]
  Call Extruder(212.04640)
  MoveL 3635 to (241.06, 52.75, 59.84) mm, rotated rx -180 ry 0 rz 180 deg; joints [-19.368, 14.547, 54.957, 45.113, 27.91, -41.578]
  MoveL 3636 to (241.06, 52.75, 59.84) mm, rotated rx -180 ry 0 rz 180 deg; joints [-19.368, 14.547, 54.957, 45.113, 27.91, -41.578]
  Call Extruder(212.34184)
  MoveL 3637 to (241.11, 53.34, 59.84) mm, rotated rx -180 ry 0 rz 180 deg; joints [-19.428, 14.594, 54.898, 45.192, 27.959, -41.645]
  MoveL 3638 to (241.11, 53.34, 59.84) mm, rotated rx -180 ry 0 rz 180 deg; joints [-19.428, 14.594, 54.898, 45.192, 27.959, -41.645]
  Call Extruder(212.63595)
  MoveL 3639 to (241.15, 53.93, 59.84) mm, rotated rx -180 ry 0 rz 180 deg; joints [-19.488, 14.641, 54.838, 45.271, 28.007, -41.71]
  MoveL 3640 to (241.15, 53.93, 59.84) mm, rotated rx -180 ry 0 rz 180 deg; joints [-19.488, 14.641, 54.838, 45.271, 28.007, -41.71]
  Call Extruder(212.92873)
  MoveL 3641 to (241.2, 54.52, 59.84) mm, rotated rx 180 ry 0 rz 180 deg; joints [-19.548, 14.688, 54.779, 45.35, 28.056, -41.776]
  MoveL 3642 to (241.2, 54.52, 59.84) mm, rotated rx 180 ry 0 rz 180 deg; joints [-19.548, 14.688, 54.779, 45.35, 28.056, -41.776]
  Call Extruder(213.50218)
  MoveL 3643 to (241.25, 55.68, 59.84) mm, rotated rx 180 ry 0 rz 180 deg; joints [-19.668, 14.773, 54.671, 45.51, 28.152, -41.909]
  MoveL 3644 to (241.25, 55.68, 59.84) mm, rotated rx 180 ry 0 rz 180 deg; joints [-19.668, 14.773, 54.671, 45.51, 28.152, -41.909]
  Call Extruder(214.21601)
  MoveL 3645 to (241.29, 57.14, 59.84) mm, rotated rx 180 ry 0 rz 180 deg; joints [-19.819, 14.876, 54.54, 45.709, 28.272, -42.075]
  Call Extruder(256.28089)
  MoveL 3646 to (241.29, 142.86, 59.84) mm, rotated rx 180 ry 0 rz 180 deg; joints [-28.232, 22.422, 44.423, 53.782, 35.898, -47.883]
  Call Extruder(256.70932)
  MoveL 3647 to (241.27, 143.73, 59.84) mm, rotated rx -180 ry 0 rz 180 deg; joints [-28.313, 22.518, 44.287, 53.83, 35.981, -47.903]
  MoveL 3648 to (241.27, 143.73, 59.84) mm, rotated rx -180 ry 0 rz 180 deg; joints [-28.313, 22.518, 44.287, 53.83, 35.981, -47.903]
  Call Extruder(257.28277)
  MoveL 3649 to (241.22, 144.9, 59.84) mm, rotated rx 180 ry 0 rz 180 deg; joints [-28.421, 22.643, 44.11, 53.896, 36.092, -47.932]
  MoveL 3650 to (241.22, 144.9, 59.84) mm, rotated rx 180 ry 0 rz 180 deg; joints [-28.421, 22.643, 44.11, 53.896, 36.092, -47.932]
  Call Extruder(257.71711)
  MoveL 3651 to (241.18, 145.77, 59.84) mm, rotated rx 180 ry 0 rz -180 deg; joints [-28.503, 22.735, 43.98, 53.947, 36.176, -47.955]
  MoveL 3652 to (241.18, 145.77, 59.84) mm, rotated rx 180 ry 0 rz -180 deg; joints [-28.503, 22.735, 43.98, 53.947, 36.176, -47.955]
  Call Extruder(258.01122)
  MoveL 3653 to (241.13, 146.36, 59.84) mm, rotated rx 180 ry 0 rz 180 deg; joints [-28.559, 22.793, 43.897, 53.983, 36.232, -47.972]
  MoveL 3654 to (241.13, 146.36, 59.84) mm, rotated rx 180 ry 0 rz 180 deg; joints [-28.559, 22.793, 43.897, 53.983, 36.232, -47.972]
  Call Extruder(258.30666)
  MoveL 3655 to (241.09, 146.95, 59.84) mm, rotated rx -180 ry 0 rz 180 deg; joints [-28.615, 22.853, 43.813, 54.019, 36.288, -47.989]
  MoveL 3656 to (241.09, 146.95, 59.84) mm, rotated rx -180 ry 0 rz 180 deg; joints [-28.615, 22.853, 43.813, 54.019, 36.288, -47.989]
  Call Extruder(258.55291)
  MoveL 3657 to (241.04, 147.44, 59.84) mm, rotated rx 180 ry 0 rz -180 deg; joints [-28.662, 22.9, 43.745, 54.049, 36.335, -48.004]
  MoveL 3658 to (241.04, 147.44, 59.84) mm, rotated rx 180 ry 0 rz -180 deg; joints [-28.662, 22.9, 43.745, 54.049, 36.335, -48.004]
  Call Extruder(258.74962)
  MoveL 3659 to (240.99, 147.83, 59.84) mm, rotated rx -180 ry 0 rz 180 deg; joints [-28.7, 22.936, 43.694, 54.075, 36.371, -48.018]
  MoveL 3660 to (240.99, 147.83, 59.84) mm, rotated rx -180 ry 0 rz 180 deg; joints [-28.7, 22.936, 43.694, 54.075, 36.371, -48.018]
  Call Extruder(258.94719)
  MoveL 3661 to (240.95, 148.22, 59.84) mm, rotated rx 180 ry 0 rz 180 deg; joints [-28.737, 22.972, 43.643, 54.101, 36.408, -48.031]
  MoveL 3662 to (240.95, 148.22, 59.84) mm, rotated rx 180 ry 0 rz 180 deg; joints [-28.737, 22.972, 43.643, 54.101, 36.408, -48.031]
  Call Extruder(259.14563)
  MoveL 3663 to (240.9, 148.6, 59.84) mm, rotated rx -180 ry 0 rz -180 deg; joints [-28.774, 23.008, 43.592, 54.126, 36.445, -48.044]
  MoveL 3664 to (240.9, 148.6, 59.84) mm, rotated rx -180 ry 0 rz -180 deg; joints [-28.774, 23.008, 43.592, 54.126, 36.445, -48.044]
  Call Extruder(259.34494)
  MoveL 3665 to (240.86, 148.99, 59.84) mm, rotated rx 180 ry 0 rz 180 deg; joints [-28.812, 23.044, 43.541, 54.151, 36.482, -48.057]
  MoveL 3666 to (240.86, 148.99, 59.84) mm, rotated rx 180 ry 0 rz 180 deg; joints [-28.812, 23.044, 43.541, 54.151, 36.482, -48.057]
  Call Extruder(259.50377)
  MoveL 3667 to (240.81, 149.3, 59.84) mm, rotated rx 180 ry 0 rz 180 deg; joints [-28.842, 23.07, 43.503, 54.173, 36.511, -48.069]
  MoveL 3668 to (240.81, 149.3, 59.84) mm, rotated rx 180 ry 0 rz 180 deg; joints [-28.842, 23.07, 43.503, 54.173, 36.511, -48.069]
  Call Extruder(259.66333)
  MoveL 3669 to (240.76, 149.6, 59.84) mm, rotated rx -180 ry 0 rz -180 deg; joints [-28.872, 23.096, 43.467, 54.195, 36.539, -48.082]
  MoveL 3670 to (240.76, 149.6, 59.84) mm, rotated rx -180 ry 0 rz -180 deg; joints [-28.872, 23.096, 43.467, 54.195, 36.539, -48.082]
  Call Extruder(259.82362)
  MoveL 3671 to (240.71, 149.91, 59.84) mm, rotated rx 180 ry 0 rz -180 deg; joints [-28.902, 23.122, 43.429, 54.216, 36.568, -48.093]
  MoveL 3672 to (240.71, 149.91, 59.84) mm, rotated rx 180 ry 0 rz -180 deg; joints [-28.902, 23.122, 43.429, 54.216, 36.568, -48.093]
  Call Extruder(259.98464)
  MoveL 3673 to (240.66, 150.21, 59.84) mm, rotated rx -180 ry 0 rz 180 deg; joints [-28.932, 23.148, 43.392, 54.238, 36.597, -48.105]
  MoveL 3674 to (240.66, 150.21, 59.84) mm, rotated rx -180 ry 0 rz 180 deg; joints [-28.932, 23.148, 43.392, 54.238, 36.597, -48.105]
  Call Extruder(260.14638)
  MoveL 3675 to (240.61, 150.52, 59.84) mm, rotated rx 180 ry 0 rz 180 deg; joints [-28.962, 23.174, 43.355, 54.259, 36.626, -48.117]
  MoveL 3676 to (240.61, 150.52, 59.84) mm, rotated rx 180 ry 0 rz 180 deg; joints [-28.962, 23.174, 43.355, 54.259, 36.626, -48.117]
  Call Extruder(260.30885)
  MoveL 3677 to (240.57, 150.83, 59.84) mm, rotated rx 180 ry 0 rz 180 deg; joints [-28.993, 23.2, 43.317, 54.281, 36.655, -48.129]
  MoveL 3678 to (240.57, 150.83, 59.84) mm, rotated rx 180 ry 0 rz 180 deg; joints [-28.993, 23.2, 43.317, 54.281, 36.655, -48.129]
  Call Extruder(260.44278)
  MoveL 3679 to (240.52, 151.08, 59.84) mm, rotated rx -180 ry 0 rz 180 deg; joints [-29.017, 23.219, 43.29, 54.3, 36.679, -48.14]
  MoveL 3680 to (240.52, 151.08, 59.84) mm, rotated rx -180 ry 0 rz 180 deg; joints [-29.017, 23.219, 43.29, 54.3, 36.679, -48.14]
  Call Extruder(260.57732)
  MoveL 3681 to (240.47, 151.32, 59.84) mm, rotated rx 180 ry 0 rz 180 deg; joints [-29.043, 23.238, 43.262, 54.319, 36.702, -48.151]
  MoveL 3682 to (240.47, 151.32, 59.84) mm, rotated rx 180 ry 0 rz 180 deg; joints [-29.043, 23.238, 43.262, 54.319, 36.702, -48.151]
  Call Extruder(260.71246)
  MoveL 3683 to (240.42, 151.57, 59.84) mm, rotated rx 180 ry 0 rz 180 deg; joints [-29.067, 23.258, 43.235, 54.338, 36.725, -48.162]
  MoveL 3684 to (240.42, 151.57, 59.84) mm, rotated rx 180 ry 0 rz 180 deg; joints [-29.067, 23.258, 43.235, 54.338, 36.725, -48.162]
  Call Extruder(260.84822)
  MoveL 3685 to (240.37, 151.82, 59.84) mm, rotated rx 180 ry 0 rz 180 deg; joints [-29.092, 23.277, 43.207, 54.356, 36.749, -48.173]
  MoveL 3686 to (240.37, 151.82, 59.84) mm, rotated rx 180 ry 0 rz 180 deg; joints [-29.092, 23.277, 43.207, 54.356, 36.749, -48.173]
  Call Extruder(260.98459)
  MoveL 3687 to (240.32, 152.07, 59.84) mm, rotated rx 180 ry 0 rz 180 deg; joints [-29.117, 23.296, 43.18, 54.375, 36.772, -48.184]
  MoveL 3688 to (240.32, 152.07, 59.84) mm, rotated rx 180 ry 0 rz 180 deg; joints [-29.117, 23.296, 43.18, 54.375, 36.772, -48.184]
  Call Extruder(261.12157)
  MoveL 3689 to (240.27, 152.32, 59.84) mm, rotated rx 180 ry 0 rz 180 deg; joints [-29.142, 23.316, 43.152, 54.394, 36.796, -48.195]
  MoveL 3690 to (240.27, 152.32, 59.84) mm, rotated rx 180 ry 0 rz 180 deg; joints [-29.142, 23.316, 43.152, 54.394, 36.796, -48.195]
  Call Extruder(261.25915)
  MoveL 3691 to (240.22, 152.57, 59.84) mm, rotated rx 180 ry 0 rz 180 deg; joints [-29.167, 23.335, 43.124, 54.412, 36.819, -48.206]
  MoveL 3692 to (240.22, 152.57, 59.84) mm, rotated rx 180 ry 0 rz 180 deg; joints [-29.167, 23.335, 43.124, 54.412, 36.819, -48.206]
  Call Extruder(261.37285)
  MoveL 3693 to (240.17, 152.77, 59.84) mm, rotated rx -180 ry 0 rz 180 deg; joints [-29.188, 23.351, 43.102, 54.428, 36.839, -48.216]
  MoveL 3694 to (240.17, 152.77, 59.84) mm, rotated rx -180 ry 0 rz 180 deg; joints [-29.188, 23.351, 43.102, 54.428, 36.839, -48.216]
  Call Extruder(261.48700)
  MoveL 3695 to (240.13, 152.98, 59.84) mm, rotated rx 180 ry 0 rz 180 deg; joints [-29.209, 23.366, 43.081, 54.444, 36.858, -48.225]
  MoveL 3696 to (240.13, 152.98, 59.84) mm, rotated rx 180 ry 0 rz 180 deg; joints [-29.209, 23.366, 43.081, 54.444, 36.858, -48.225]
  Call Extruder(261.60161)
  MoveL 3697 to (240.08, 153.18, 59.84) mm, rotated rx 180 ry 0 rz 180 deg; joints [-29.229, 23.381, 43.059, 54.46, 36.877, -48.235]
  MoveL 3698 to (240.08, 153.18, 59.84) mm, rotated rx 180 ry 0 rz 180 deg; joints [-29.229, 23.381, 43.059, 54.46, 36.877, -48.235]
  Call Extruder(261.71666)
  MoveL 3699 to (240.04, 153.39, 59.84) mm, rotated rx -180 ry 0 rz 180 deg; joints [-29.25, 23.396, 43.037, 54.476, 36.896, -48.244]
  MoveL 3700 to (240.04, 153.39, 59.84) mm, rotated rx -180 ry 0 rz 180 deg; joints [-29.25, 23.396, 43.037, 54.476, 36.896, -48.244]
  Call Extruder(261.83888)
  MoveL 3701 to (239.98, 153.6, 59.84) mm, rotated rx -180 ry 0 rz -180 deg; joints [-29.272, 23.41, 43.017, 54.494, 36.916, -48.255]
  MoveL 3702 to (239.98, 153.6, 59.84) mm, rotated rx -180 ry 0 rz -180 deg; joints [-29.272, 23.41, 43.017, 54.494, 36.916, -48.255]
  Call Extruder(261.96855)
  MoveL 3703 to (239.92, 153.82, 59.84) mm, rotated rx -180 ry 0 rz 180 deg; joints [-29.296, 23.422, 42.999, 54.514, 36.937, -48.269]
  MoveL 3704 to (239.92, 153.82, 59.84) mm, rotated rx -180 ry 0 rz 180 deg; joints [-29.296, 23.422, 42.999, 54.514, 36.937, -48.269]
  Call Extruder(262.09877)
  MoveL 3705 to (239.85, 154.05, 59.84) mm, rotated rx 180 ry 0 rz 180 deg; joints [-29.319, 23.435, 42.981, 54.534, 36.958, -48.282]
  MoveL 3706 to (239.85, 154.05, 59.84) mm, rotated rx 180 ry 0 rz 180 deg; joints [-29.319, 23.435, 42.981, 54.534, 36.958, -48.282]
  Call Extruder(262.22956)
  MoveL 3707 to (239.78, 154.27, 59.84) mm, rotated rx 180 ry 0 rz 180 deg; joints [-29.343, 23.448, 42.963, 54.554, 36.978, -48.296]
  MoveL 3708 to (239.78, 154.27, 59.84) mm, rotated rx 180 ry 0 rz 180 deg; joints [-29.343, 23.448, 42.963, 54.554, 36.978, -48.296]
  Call Extruder(262.36092)
  MoveL 3709 to (239.71, 154.49, 59.84) mm, rotated rx 180 ry 0 rz 180 deg; joints [-29.366, 23.46, 42.945, 54.574, 36.999, -48.309]
  MoveL 3710 to (239.71, 154.49, 59.84) mm, rotated rx 180 ry 0 rz 180 deg; joints [-29.366, 23.46, 42.945, 54.574, 36.999, -48.309]
  Call Extruder(262.47282)
  MoveL 3711 to (239.65, 154.68, 59.84) mm, rotated rx -180 ry 0 rz 180 deg; joints [-29.386, 23.47, 42.931, 54.592, 37.017, -48.321]
  MoveL 3712 to (239.65, 154.68, 59.84) mm, rotated rx -180 ry 0 rz 180 deg; joints [-29.386, 23.47, 42.931, 54.592, 37.017, -48.321]
  Call Extruder(262.58516)
  MoveL 3713 to (239.59, 154.87, 59.84) mm, rotated rx -180 ry 0 rz 180 deg; joints [-29.406, 23.48, 42.916, 54.609, 37.034, -48.333]
  MoveL 3714 to (239.59, 154.87, 59.84) mm, rotated rx -180 ry 0 rz 180 deg; joints [-29.406, 23.48, 42.916, 54.609, 37.034, -48.333]
  Call Extruder(262.69795)
  MoveL 3715 to (239.53, 155.06, 59.84) mm, rotated rx -180 ry 0 rz 180 deg; joints [-29.426, 23.49, 42.903, 54.627, 37.051, -48.345]
  MoveL 3716 to (239.53, 155.06, 59.84) mm, rotated rx -180 ry 0 rz 180 deg; joints [-29.426, 23.49, 42.903, 54.627, 37.051, -48.345]
  Call Extruder(262.81119)
  MoveL 3717 to (239.47, 155.25, 59.84) mm, rotated rx -180 ry 0 rz 180 deg; joints [-29.446, 23.5, 42.888, 54.644, 37.069, -48.357]
  MoveL 3718 to (239.47, 155.25, 59.84) mm, rotated rx -180 ry 0 rz 180 deg; joints [-29.446, 23.5, 42.888, 54.644, 37.069, -48.357]
  Call Extruder(262.92487)
  MoveL 3719 to (239.41, 155.44, 59.84) mm, rotated rx 180 ry 0 rz -180 deg; joints [-29.466, 23.51, 42.874, 54.662, 37.086, -48.368]
  MoveL 3720 to (239.41, 155.44, 59.84) mm, rotated rx 180 ry 0 rz -180 deg; joints [-29.466, 23.51, 42.874, 54.662, 37.086, -48.368]
  Call Extruder(263.10683)
  MoveL 3721 to (239.29, 155.73, 59.84) mm, rotated rx -180 ry 0 rz -180 deg; joints [-29.499, 23.519, 42.86, 54.693, 37.113, -48.391]
  MoveL 3722 to (239.29, 155.73, 59.84) mm, rotated rx -180 ry 0 rz -180 deg; joints [-29.499, 23.519, 42.86, 54.693, 37.113, -48.391]
  Call Extruder(263.28954)
  MoveL 3723 to (239.16, 156.02, 59.84) mm, rotated rx -180 ry 0 rz 180 deg; joints [-29.531, 23.529, 42.847, 54.724, 37.14, -48.414]
  MoveL 3724 to (239.16, 156.02, 59.84) mm, rotated rx -180 ry 0 rz 180 deg; joints [-29.531, 23.529, 42.847, 54.724, 37.14, -48.414]
  Call Extruder(263.45997)
  MoveL 3725 to (239.05, 156.29, 59.84) mm, rotated rx -180 ry 0 rz 180 deg; joints [-29.561, 23.537, 42.834, 54.753, 37.164, -48.435]
  MoveL 3726 to (239.05, 156.29, 59.84) mm, rotated rx -180 ry 0 rz 180 deg; joints [-29.561, 23.537, 42.834, 54.753, 37.164, -48.435]
  Call Extruder(263.61798)
  MoveL 3727 to (238.94, 156.54, 59.84) mm, rotated rx 180 ry 0 rz -180 deg; joints [-29.589, 23.545, 42.824, 54.78, 37.187, -48.455]
  MoveL 3728 to (238.94, 156.54, 59.84) mm, rotated rx 180 ry 0 rz -180 deg; joints [-29.589, 23.545, 42.824, 54.78, 37.187, -48.455]
  Call Extruder(263.77659)
  MoveL 3729 to (238.84, 156.79, 59.84) mm, rotated rx -180 ry 0 rz 180 deg; joints [-29.617, 23.553, 42.813, 54.807, 37.21, -48.475]
  MoveL 3730 to (238.84, 156.79, 59.84) mm, rotated rx -180 ry 0 rz 180 deg; joints [-29.617, 23.553, 42.813, 54.807, 37.21, -48.475]
  Call Extruder(263.98276)
  MoveL 3731 to (238.66, 157.09, 59.84) mm, rotated rx 180 ry 0 rz 180 deg; joints [-29.653, 23.552, 42.813, 54.847, 37.237, -48.507]
  MoveL 3732 to (238.66, 157.09, 59.84) mm, rotated rx 180 ry 0 rz 180 deg; joints [-29.653, 23.552, 42.813, 54.847, 37.237, -48.507]
  Call Extruder(264.18971)
  MoveL 3733 to (238.49, 157.4, 59.84) mm, rotated rx -180 ry 0 rz 180 deg; joints [-29.689, 23.552, 42.814, 54.887, 37.263, -48.539]
  MoveL 3734 to (238.49, 157.4, 59.84) mm, rotated rx -180 ry 0 rz 180 deg; joints [-29.689, 23.552, 42.814, 54.887, 37.263, -48.539]
  Call Extruder(264.39743)
  MoveL 3735 to (238.31, 157.7, 59.84) mm, rotated rx -180 ry 0 rz 180 deg; joints [-29.725, 23.551, 42.815, 54.926, 37.291, -48.57]
  MoveL 3736 to (238.31, 157.7, 59.84) mm, rotated rx -180 ry 0 rz 180 deg; joints [-29.725, 23.551, 42.815, 54.926, 37.291, -48.57]
  Call Extruder(264.60594)
  MoveL 3737 to (238.14, 158.01, 59.84) mm, rotated rx 180 ry 0 rz 180 deg; joints [-29.761, 23.551, 42.815, 54.966, 37.318, -48.602]
  MoveL 3738 to (238.14, 158.01, 59.84) mm, rotated rx 180 ry 0 rz 180 deg; joints [-29.761, 23.551, 42.815, 54.966, 37.318, -48.602]
  Call Extruder(264.78548)
  MoveL 3739 to (237.96, 158.25, 59.84) mm, rotated rx 180 ry 0 rz -180 deg; joints [-29.792, 23.543, 42.827, 55.003, 37.339, -48.633]
  MoveL 3740 to (237.96, 158.25, 59.84) mm, rotated rx 180 ry 0 rz -180 deg; joints [-29.792, 23.543, 42.827, 55.003, 37.339, -48.633]
  Call Extruder(265.11889)
  MoveL 3741 to (237.63, 158.7, 59.84) mm, rotated rx 180 ry 0 rz 180 deg; joints [-29.849, 23.528, 42.848, 55.073, 37.378, -48.692]
  MoveL 3742 to (237.63, 158.7, 59.84) mm, rotated rx 180 ry 0 rz 180 deg; joints [-29.849, 23.528, 42.848, 55.073, 37.378, -48.692]
  Call Extruder(265.45348)
  MoveL 3743 to (237.3, 159.15, 59.84) mm, rotated rx 180 ry 0 rz 180 deg; joints [-29.907, 23.513, 42.87, 55.142, 37.417, -48.75]
  Call Extruder(266.28143)
  MoveL 3744 to (236.39, 160.19, 59.84) mm, rotated rx 180 ry 0 rz 180 deg; joints [-30.046, 23.445, 42.967, 55.325, 37.506, -48.91]
  Call Extruder(267.10937)
  MoveL 3745 to (235.35, 161.1, 59.84) mm, rotated rx 180 ry 0 rz -180 deg; joints [-30.182, 23.335, 43.124, 55.521, 37.581, -49.089]
  Call Extruder(267.27668)
  MoveL 3746 to (235.13, 161.27, 59.84) mm, rotated rx 180 ry 0 rz 180 deg; joints [-30.208, 23.307, 43.165, 55.562, 37.594, -49.128]
  MoveL 3747 to (235.13, 161.27, 59.84) mm, rotated rx 180 ry 0 rz 180 deg; joints [-30.208, 23.307, 43.165, 55.562, 37.594, -49.128]
  Call Extruder(267.61010)
  MoveL 3748 to (234.68, 161.59, 59.84) mm, rotated rx 180 ry 0 rz 180 deg; joints [-30.261, 23.251, 43.245, 55.644, 37.62, -49.205]
  MoveL 3749 to (234.68, 161.59, 59.84) mm, rotated rx 180 ry 0 rz 180 deg; joints [-30.261, 23.251, 43.245, 55.644, 37.62, -49.205]
  Call Extruder(267.94234)
  MoveL 3750 to (234.23, 161.92, 59.84) mm, rotated rx -180 ry 0 rz 180 deg; joints [-30.314, 23.195, 43.324, 55.727, 37.647, -49.282]
  MoveL 3751 to (234.23, 161.92, 59.84) mm, rotated rx -180 ry 0 rz 180 deg; joints [-30.314, 23.195, 43.324, 55.727, 37.647, -49.282]
  Call Extruder(268.06000)
  MoveL 3752 to (234.05, 162.02, 59.84) mm, rotated rx -180 ry 0 rz 180 deg; joints [-30.331, 23.171, 43.359, 55.757, 37.654, -49.311]
  MoveL 3753 to (234.05, 162.02, 59.84) mm, rotated rx -180 ry 0 rz 180 deg; joints [-30.331, 23.171, 43.359, 55.757, 37.654, -49.311]
  Call Extruder(268.26773)
  MoveL 3754 to (233.75, 162.2, 59.84) mm, rotated rx 180 ry 0 rz 180 deg; joints [-30.363, 23.128, 43.42, 55.81, 37.668, -49.363]
  MoveL 3755 to (233.75, 162.2, 59.84) mm, rotated rx 180 ry 0 rz 180 deg; joints [-30.363, 23.128, 43.42, 55.81, 37.668, -49.363]
  Call Extruder(268.47467)
  MoveL 3756 to (233.45, 162.37, 59.84) mm, rotated rx 180 ry 0 rz 180 deg; joints [-30.394, 23.085, 43.481, 55.863, 37.681, -49.414]
  MoveL 3757 to (233.45, 162.37, 59.84) mm, rotated rx 180 ry 0 rz 180 deg; joints [-30.394, 23.085, 43.481, 55.863, 37.681, -49.414]
  Call Extruder(268.68084)
  MoveL 3758 to (233.14, 162.55, 59.84) mm, rotated rx -180 ry 0 rz 180 deg; joints [-30.426, 23.042, 43.542, 55.916, 37.695, -49.466]
  MoveL 3759 to (233.14, 162.55, 59.84) mm, rotated rx -180 ry 0 rz 180 deg; joints [-30.426, 23.042, 43.542, 55.916, 37.695, -49.466]
  Call Extruder(268.86251)
  MoveL 3760 to (232.87, 162.69, 59.84) mm, rotated rx 180 ry 0 rz 180 deg; joints [-30.453, 23.001, 43.601, 55.964, 37.706, -49.512]
  MoveL 3761 to (232.87, 162.69, 59.84) mm, rotated rx 180 ry 0 rz 180 deg; joints [-30.453, 23.001, 43.601, 55.964, 37.706, -49.512]
  Call Extruder(269.02049)
  MoveL 3762 to (232.62, 162.8, 59.84) mm, rotated rx 180 ry 0 rz -180 deg; joints [-30.476, 22.962, 43.657, 56.006, 37.714, -49.554]
  MoveL 3763 to (232.62, 162.8, 59.84) mm, rotated rx 180 ry 0 rz -180 deg; joints [-30.476, 22.962, 43.657, 56.006, 37.714, -49.554]
  Call Extruder(269.17786)
  MoveL 3764 to (232.37, 162.91, 59.84) mm, rotated rx 180 ry 0 rz 180 deg; joints [-30.498, 22.922, 43.713, 56.048, 37.722, -49.595]
  MoveL 3765 to (232.37, 162.91, 59.84) mm, rotated rx 180 ry 0 rz 180 deg; joints [-30.498, 22.922, 43.713, 56.048, 37.722, -49.595]
  Call Extruder(269.36060)
  MoveL 3766 to (232.07, 163.03, 59.84) mm, rotated rx 180 ry 0 rz 180 deg; joints [-30.524, 22.876, 43.78, 56.097, 37.731, -49.644]
  MoveL 3767 to (232.07, 163.03, 59.84) mm, rotated rx 180 ry 0 rz 180 deg; joints [-30.524, 22.876, 43.78, 56.097, 37.731, -49.644]
  Call Extruder(269.54259)
  MoveL 3768 to (231.78, 163.15, 59.84) mm, rotated rx -180 ry 0 rz -180 deg; joints [-30.551, 22.829, 43.846, 56.145, 37.74, -49.692]
  MoveL 3769 to (231.78, 163.15, 59.84) mm, rotated rx -180 ry 0 rz -180 deg; joints [-30.551, 22.829, 43.846, 56.145, 37.74, -49.692]
  Call Extruder(269.68992)
  MoveL 3770 to (231.54, 163.24, 59.84) mm, rotated rx 180 ry 0 rz 180 deg; joints [-30.571, 22.79, 43.902, 56.185, 37.746, -49.732]
  MoveL 3771 to (231.54, 163.24, 59.84) mm, rotated rx 180 ry 0 rz 180 deg; joints [-30.571, 22.79, 43.902, 56.185, 37.746, -49.732]
  Call Extruder(269.80315)
  MoveL 3772 to (231.35, 163.3, 59.84) mm, rotated rx 180 ry 0 rz 180 deg; joints [-30.587, 22.758, 43.947, 56.216, 37.751, -49.763]
  MoveL 3773 to (231.35, 163.3, 59.84) mm, rotated rx 180 ry 0 rz 180 deg; joints [-30.587, 22.758, 43.947, 56.216, 37.751, -49.763]
  Call Extruder(269.91592)
  MoveL 3774 to (231.17, 163.36, 59.84) mm, rotated rx 180 ry 0 rz 180 deg; joints [-30.602, 22.726, 43.993, 56.246, 37.755, -49.794]
  MoveL 3775 to (231.17, 163.36, 59.84) mm, rotated rx 180 ry 0 rz 180 deg; joints [-30.602, 22.726, 43.993, 56.246, 37.755, -49.794]
  Call Extruder(270.02826)
  MoveL 3776 to (230.98, 163.42, 59.84) mm, rotated rx 180 ry 0 rz 180 deg; joints [-30.618, 22.694, 44.038, 56.277, 37.759, -49.825]
  MoveL 3777 to (230.98, 163.42, 59.84) mm, rotated rx 180 ry 0 rz 180 deg; joints [-30.618, 22.694, 44.038, 56.277, 37.759, -49.825]
  Call Extruder(270.14014)
  MoveL 3778 to (230.79, 163.48, 59.84) mm, rotated rx 180 ry 0 rz 180 deg; joints [-30.633, 22.662, 44.083, 56.307, 37.764, -49.856]
  MoveL 3779 to (230.79, 163.48, 59.84) mm, rotated rx 180 ry 0 rz 180 deg; joints [-30.633, 22.662, 44.083, 56.307, 37.764, -49.856]
  Call Extruder(270.26155)
  MoveL 3780 to (230.58, 163.55, 59.84) mm, rotated rx 180 ry 0 rz 180 deg; joints [-30.65, 22.627, 44.133, 56.341, 37.768, -49.89]
  MoveL 3781 to (230.58, 163.55, 59.84) mm, rotated rx 180 ry 0 rz 180 deg; joints [-30.65, 22.627, 44.133, 56.341, 37.768, -49.89]
  Call Extruder(270.39236)
  MoveL 3782 to (230.36, 163.61, 59.84) mm, rotated rx 180 ry 0 rz 180 deg; joints [-30.668, 22.588, 44.187, 56.377, 37.773, -49.927]
  MoveL 3783 to (230.36, 163.61, 59.84) mm, rotated rx 180 ry 0 rz 180 deg; joints [-30.668, 22.588, 44.187, 56.377, 37.773, -49.927]
  Call Extruder(270.52261)
  MoveL 3784 to (230.14, 163.68, 59.84) mm, rotated rx 180 ry 0 rz -180 deg; joints [-30.685, 22.55, 44.241, 56.413, 37.778, -49.963]
  MoveL 3785 to (230.14, 163.68, 59.84) mm, rotated rx 180 ry 0 rz -180 deg; joints [-30.685, 22.55, 44.241, 56.413, 37.778, -49.963]
  Call Extruder(270.65229)
  MoveL 3786 to (229.91, 163.75, 59.84) mm, rotated rx 180 ry 0 rz 180 deg; joints [-30.703, 22.512, 44.296, 56.448, 37.783, -50]
  MoveL 3787 to (229.91, 163.75, 59.84) mm, rotated rx 180 ry 0 rz 180 deg; joints [-30.703, 22.512, 44.296, 56.448, 37.783, -50]
  Call Extruder(270.78141)
  MoveL 3788 to (229.69, 163.82, 59.84) mm, rotated rx 180 ry 0 rz 180 deg; joints [-30.721, 22.474, 44.35, 56.484, 37.788, -50.036]
  MoveL 3789 to (229.69, 163.82, 59.84) mm, rotated rx 180 ry 0 rz 180 deg; joints [-30.721, 22.474, 44.35, 56.484, 37.788, -50.036]
  Call Extruder(270.89648)
  MoveL 3790 to (229.48, 163.86, 59.84) mm, rotated rx 180 ry 0 rz -180 deg; joints [-30.736, 22.437, 44.402, 56.516, 37.791, -50.069]
  MoveL 3791 to (229.48, 163.86, 59.84) mm, rotated rx 180 ry 0 rz -180 deg; joints [-30.736, 22.437, 44.402, 56.516, 37.791, -50.069]
  Call Extruder(271.01110)
  MoveL 3792 to (229.28, 163.91, 59.84) mm, rotated rx -180 ry 0 rz 180 deg; joints [-30.751, 22.4, 44.454, 56.548, 37.794, -50.102]
  MoveL 3793 to (229.28, 163.91, 59.84) mm, rotated rx -180 ry 0 rz 180 deg; joints [-30.751, 22.4, 44.454, 56.548, 37.794, -50.102]
  Call Extruder(271.12527)
  MoveL 3794 to (229.08, 163.95, 59.84) mm, rotated rx 180 ry 0 rz -180 deg; joints [-30.766, 22.363, 44.506, 56.58, 37.797, -50.135]
  MoveL 3795 to (229.08, 163.95, 59.84) mm, rotated rx 180 ry 0 rz -180 deg; joints [-30.766, 22.363, 44.506, 56.58, 37.797, -50.135]
  Call Extruder(271.23899)
  MoveL 3796 to (228.87, 164, 59.84) mm, rotated rx 180 ry 0 rz 180 deg; joints [-30.781, 22.326, 44.558, 56.612, 37.8, -50.168]
  MoveL 3797 to (228.87, 164, 59.84) mm, rotated rx 180 ry 0 rz 180 deg; joints [-30.781, 22.326, 44.558, 56.612, 37.8, -50.168]
  Call Extruder(271.36441)
  MoveL 3798 to (228.65, 164.04, 59.84) mm, rotated rx 180 ry 0 rz -180 deg; joints [-30.797, 22.286, 44.615, 56.647, 37.803, -50.204]
  MoveL 3799 to (228.65, 164.04, 59.84) mm, rotated rx 180 ry 0 rz -180 deg; joints [-30.797, 22.286, 44.615, 56.647, 37.803, -50.204]
  Call Extruder(271.50139)
  MoveL 3800 to (228.4, 164.09, 59.84) mm, rotated rx 180 ry 0 rz 180 deg; joints [-30.815, 22.24, 44.679, 56.685, 37.807, -50.244]
  MoveL 3801 to (228.4, 164.09, 59.84) mm, rotated rx 180 ry 0 rz 180 deg; joints [-30.815, 22.24, 44.679, 56.685, 37.807, -50.244]
  Call Extruder(271.63776)
  MoveL 3802 to (228.15, 164.14, 59.84) mm, rotated rx 180 ry 0 rz -180 deg; joints [-30.832, 22.195, 44.743, 56.724, 37.81, -50.284]
  MoveL 3803 to (228.15, 164.14, 59.84) mm, rotated rx 180 ry 0 rz -180 deg; joints [-30.832, 22.195, 44.743, 56.724, 37.81, -50.284]
  Call Extruder(271.77351)
  MoveL 3804 to (227.9, 164.19, 59.84) mm, rotated rx -180 ry 0 rz -180 deg; joints [-30.85, 22.15, 44.807, 56.762, 37.814, -50.324]
  MoveL 3805 to (227.9, 164.19, 59.84) mm, rotated rx -180 ry 0 rz -180 deg; joints [-30.85, 22.15, 44.807, 56.762, 37.814, -50.324]
  Call Extruder(271.90866)
  MoveL 3806 to (227.65, 164.24, 59.84) mm, rotated rx -180 ry 0 rz 180 deg; joints [-30.868, 22.105, 44.87, 56.8, 37.817, -50.363]
  MoveL 3807 to (227.65, 164.24, 59.84) mm, rotated rx -180 ry 0 rz 180 deg; joints [-30.868, 22.105, 44.87, 56.8, 37.817, -50.363]
  Call Extruder(272.04320)
  MoveL 3808 to (227.4, 164.29, 59.84) mm, rotated rx 180 ry 0 rz 180 deg; joints [-30.886, 22.06, 44.933, 56.839, 37.821, -50.403]
  MoveL 3809 to (227.4, 164.29, 59.84) mm, rotated rx 180 ry 0 rz 180 deg; joints [-30.886, 22.06, 44.933, 56.839, 37.821, -50.403]
  Call Extruder(272.17712)
  MoveL 3810 to (227.15, 164.34, 59.84) mm, rotated rx 180 ry 0 rz 180 deg; joints [-30.903, 22.015, 44.996, 56.877, 37.825, -50.442]
  MoveL 3811 to (227.15, 164.34, 59.84) mm, rotated rx 180 ry 0 rz 180 deg; joints [-30.903, 22.015, 44.996, 56.877, 37.825, -50.442]
  Call Extruder(272.32499)
  MoveL 3812 to (226.87, 164.39, 59.84) mm, rotated rx 180 ry 0 rz -180 deg; joints [-30.923, 21.965, 45.067, 56.919, 37.828, -50.486]
  MoveL 3813 to (226.87, 164.39, 59.84) mm, rotated rx 180 ry 0 rz -180 deg; joints [-30.923, 21.965, 45.067, 56.919, 37.828, -50.486]
  Call Extruder(272.48673)
  MoveL 3814 to (226.57, 164.44, 59.84) mm, rotated rx 180 ry 0 rz 180 deg; joints [-30.943, 21.908, 45.146, 56.965, 37.832, -50.534]
  MoveL 3815 to (226.57, 164.44, 59.84) mm, rotated rx 180 ry 0 rz 180 deg; joints [-30.943, 21.908, 45.146, 56.965, 37.832, -50.534]
  Call Extruder(272.64774)
  MoveL 3816 to (226.26, 164.49, 59.84) mm, rotated rx -180 ry 0 rz 180 deg; joints [-30.964, 21.852, 45.225, 57.011, 37.836, -50.582]
  MoveL 3817 to (226.26, 164.49, 59.84) mm, rotated rx -180 ry 0 rz 180 deg; joints [-30.964, 21.852, 45.225, 57.011, 37.836, -50.582]
  Call Extruder(272.80803)
  MoveL 3818 to (225.96, 164.53, 59.84) mm, rotated rx -180 ry 0 rz 180 deg; joints [-30.985, 21.796, 45.304, 57.057, 37.839, -50.63]
  MoveL 3819 to (225.96, 164.53, 59.84) mm, rotated rx -180 ry 0 rz 180 deg; joints [-30.985, 21.796, 45.304, 57.057, 37.839, -50.63]
  Call Extruder(272.96758)
  MoveL 3820 to (225.65, 164.58, 59.84) mm, rotated rx 180 ry 0 rz 180 deg; joints [-31.006, 21.74, 45.382, 57.102, 37.843, -50.677]
  MoveL 3821 to (225.65, 164.58, 59.84) mm, rotated rx 180 ry 0 rz 180 deg; joints [-31.006, 21.74, 45.382, 57.102, 37.843, -50.677]
  Call Extruder(273.12641)
  MoveL 3822 to (225.34, 164.63, 59.84) mm, rotated rx 180 ry 0 rz 180 deg; joints [-31.027, 21.684, 45.46, 57.148, 37.847, -50.725]
  MoveL 3823 to (225.34, 164.63, 59.84) mm, rotated rx 180 ry 0 rz 180 deg; joints [-31.027, 21.684, 45.46, 57.148, 37.847, -50.725]
  Call Extruder(273.30508)
  MoveL 3824 to (225, 164.68, 59.84) mm, rotated rx 180 ry 0 rz 180 deg; joints [-31.049, 21.62, 45.55, 57.199, 37.851, -50.779]
  MoveL 3825 to (225, 164.68, 59.84) mm, rotated rx 180 ry 0 rz 180 deg; joints [-31.049, 21.62, 45.55, 57.199, 37.851, -50.779]
  Call Extruder(273.50353)
  MoveL 3826 to (224.61, 164.73, 59.84) mm, rotated rx 180 ry 0 rz 180 deg; joints [-31.074, 21.548, 45.651, 57.256, 37.855, -50.838]
  MoveL 3827 to (224.61, 164.73, 59.84) mm, rotated rx 180 ry 0 rz 180 deg; joints [-31.074, 21.548, 45.651, 57.256, 37.855, -50.838]
  Call Extruder(273.70110)
  MoveL 3828 to (224.22, 164.77, 59.84) mm, rotated rx 180 ry 0 rz 180 deg; joints [-31.1, 21.475, 45.752, 57.312, 37.859, -50.898]
  MoveL 3829 to (224.22, 164.77, 59.84) mm, rotated rx 180 ry 0 rz 180 deg; joints [-31.1, 21.475, 45.752, 57.312, 37.859, -50.898]
  Call Extruder(273.89781)
  MoveL 3830 to (223.84, 164.82, 59.84) mm, rotated rx -180 ry 0 rz 180 deg; joints [-31.125, 21.404, 45.852, 57.369, 37.863, -50.957]
  MoveL 3831 to (223.84, 164.82, 59.84) mm, rotated rx -180 ry 0 rz 180 deg; joints [-31.125, 21.404, 45.852, 57.369, 37.863, -50.957]
  Call Extruder(274.09365)
  MoveL 3832 to (223.45, 164.86, 59.84) mm, rotated rx 180 ry 0 rz 180 deg; joints [-31.15, 21.332, 45.952, 57.425, 37.868, -51.016]
  MoveL 3833 to (223.45, 164.86, 59.84) mm, rotated rx 180 ry 0 rz 180 deg; joints [-31.15, 21.332, 45.952, 57.425, 37.868, -51.016]
  Call Extruder(274.38900)
  MoveL 3834 to (222.86, 164.91, 59.84) mm, rotated rx -180 ry 0 rz 180 deg; joints [-31.186, 21.22, 46.107, 57.509, 37.872, -51.105]
  MoveL 3835 to (222.86, 164.91, 59.84) mm, rotated rx -180 ry 0 rz 180 deg; joints [-31.186, 21.22, 46.107, 57.509, 37.872, -51.105]
  Call Extruder(274.68303)
  MoveL 3836 to (222.27, 164.96, 59.84) mm, rotated rx 180 ry 0 rz 180 deg; joints [-31.222, 21.109, 46.261, 57.593, 37.877, -51.193]
  MoveL 3837 to (222.27, 164.96, 59.84) mm, rotated rx 180 ry 0 rz 180 deg; joints [-31.222, 21.109, 46.261, 57.593, 37.877, -51.193]
  Call Extruder(274.97572)
  MoveL 3838 to (221.68, 165, 59.84) mm, rotated rx 180 ry 0 rz 180 deg; joints [-31.258, 20.999, 46.415, 57.677, 37.883, -51.281]
  MoveL 3839 to (221.68, 165, 59.84) mm, rotated rx 180 ry 0 rz 180 deg; joints [-31.258, 20.999, 46.415, 57.677, 37.883, -51.281]
  Call Extruder(275.54917)
  MoveL 3840 to (220.52, 165.05, 59.84) mm, rotated rx 180 ry 0 rz 180 deg; joints [-31.326, 20.776, 46.723, 57.838, 37.89, -51.453]
  MoveL 3841 to (220.52, 165.05, 59.84) mm, rotated rx 180 ry 0 rz 180 deg; joints [-31.326, 20.776, 46.723, 57.838, 37.89, -51.453]
  Call Extruder(276.26318)
  MoveL 3842 to (219.06, 165.09, 59.84) mm, rotated rx 180 ry 0 rz 180 deg; joints [-31.409, 20.498, 47.106, 58.037, 37.9, -51.665]
  Call Extruder(393.10992)
  MoveL 3843 to (-19.06, 165.09, 59.84) mm, rotated rx 180 ry 0 rz 180 deg; joints [-51.475, -10.243, 80.711, 75.095, 54.055, -65.608]
  Call Extruder(393.53852)
  MoveL 3844 to (-19.94, 165.07, 59.84) mm, rotated rx -180 ry 0 rz 180 deg; joints [-51.582, -10.323, 80.776, 75.139, 54.156, -65.622]
  MoveL 3845 to (-19.94, 165.07, 59.84) mm, rotated rx -180 ry 0 rz 180 deg; joints [-51.582, -10.323, 80.776, 75.139, 54.156, -65.622]
  Call Extruder(394.11197)
  MoveL 3846 to (-21.1, 165.03, 59.84) mm, rotated rx -180 ry 0 rz -180 deg; joints [-51.722, -10.431, 80.864, 75.196, 54.289, -65.64]
  MoveL 3847 to (-21.1, 165.03, 59.84) mm, rotated rx -180 ry 0 rz -180 deg; joints [-51.722, -10.431, 80.864, 75.196, 54.289, -65.64]
  Call Extruder(394.54627)
  MoveL 3848 to (-21.97, 164.98, 59.84) mm, rotated rx 180 ry 0 rz 180 deg; joints [-51.827, -10.514, 80.931, 75.238, 54.389, -65.652]
  MoveL 3849 to (-21.97, 164.98, 59.84) mm, rotated rx 180 ry 0 rz 180 deg; joints [-51.827, -10.514, 80.931, 75.238, 54.389, -65.652]
  Call Extruder(394.84030)
  MoveL 3850 to (-22.56, 164.93, 59.84) mm, rotated rx 180 ry 0 rz 180 deg; joints [-51.897, -10.571, 80.977, 75.266, 54.454, -65.66]
  MoveL 3851 to (-22.56, 164.93, 59.84) mm, rotated rx 180 ry 0 rz 180 deg; joints [-51.897, -10.571, 80.977, 75.266, 54.454, -65.66]
  Call Extruder(395.13566)
  MoveL 3852 to (-23.15, 164.89, 59.84) mm, rotated rx 180 ry 0 rz 180 deg; joints [-51.966, -10.628, 81.023, 75.293, 54.521, -65.667]
  MoveL 3853 to (-23.15, 164.89, 59.84) mm, rotated rx 180 ry 0 rz 180 deg; joints [-51.966, -10.628, 81.023, 75.293, 54.521, -65.667]
  Call Extruder(395.38188)
  MoveL 3854 to (-23.64, 164.84, 59.84) mm, rotated rx 180 ry 0 rz 180 deg; joints [-52.023, -10.676, 81.062, 75.316, 54.575, -65.673]
  MoveL 3855 to (-23.64, 164.84, 59.84) mm, rotated rx 180 ry 0 rz 180 deg; joints [-52.023, -10.676, 81.062, 75.316, 54.575, -65.673]
  Call Extruder(395.57858)
  MoveL 3856 to (-24.03, 164.79, 59.84) mm, rotated rx -180 ry 0 rz 180 deg; joints [-52.067, -10.716, 81.094, 75.333, 54.617, -65.677]
  MoveL 3857 to (-24.03, 164.79, 59.84) mm, rotated rx -180 ry 0 rz 180 deg; joints [-52.067, -10.716, 81.094, 75.333, 54.617, -65.677]
  Call Extruder(395.77616)
  MoveL 3858 to (-24.42, 164.75, 59.84) mm, rotated rx -180 ry 0 rz 180 deg; joints [-52.112, -10.755, 81.126, 75.35, 54.659, -65.681]
  MoveL 3859 to (-24.42, 164.75, 59.84) mm, rotated rx -180 ry 0 rz 180 deg; joints [-52.112, -10.755, 81.126, 75.35, 54.659, -65.681]
  Call Extruder(395.97460)
  MoveL 3860 to (-24.8, 164.7, 59.84) mm, rotated rx 180 ry 0 rz 180 deg; joints [-52.156, -10.794, 81.157, 75.368, 54.702, -65.685]
  MoveL 3861 to (-24.8, 164.7, 59.84) mm, rotated rx 180 ry 0 rz 180 deg; joints [-52.156, -10.794, 81.157, 75.368, 54.702, -65.685]
  Call Extruder(396.17391)
  MoveL 3862 to (-25.19, 164.66, 59.84) mm, rotated rx 180 ry 0 rz 180 deg; joints [-52.2, -10.833, 81.189, 75.385, 54.744, -65.689]
  MoveL 3863 to (-25.19, 164.66, 59.84) mm, rotated rx 180 ry 0 rz 180 deg; joints [-52.2, -10.833, 81.189, 75.385, 54.744, -65.689]
  Call Extruder(396.33274)
  MoveL 3864 to (-25.5, 164.61, 59.84) mm, rotated rx 180 ry 0 rz 180 deg; joints [-52.235, -10.865, 81.214, 75.398, 54.777, -65.691]
  MoveL 3865 to (-25.5, 164.61, 59.84) mm, rotated rx 180 ry 0 rz 180 deg; joints [-52.235, -10.865, 81.214, 75.398, 54.777, -65.691]
  Call Extruder(396.49230)
  MoveL 3866 to (-25.8, 164.56, 59.84) mm, rotated rx 180 ry 0 rz 180 deg; joints [-52.269, -10.897, 81.24, 75.41, 54.809, -65.694]
  MoveL 3867 to (-25.8, 164.56, 59.84) mm, rotated rx 180 ry 0 rz 180 deg; joints [-52.269, -10.897, 81.24, 75.41, 54.809, -65.694]
  Call Extruder(396.65259)
  MoveL 3868 to (-26.11, 164.51, 59.84) mm, rotated rx 180 ry 0 rz -180 deg; joints [-52.303, -10.929, 81.266, 75.423, 54.842, -65.696]
  MoveL 3869 to (-26.11, 164.51, 59.84) mm, rotated rx 180 ry 0 rz -180 deg; joints [-52.303, -10.929, 81.266, 75.423, 54.842, -65.696]
  Call Extruder(396.81360)
  MoveL 3870 to (-26.41, 164.46, 59.84) mm, rotated rx 180 ry 0 rz 180 deg; joints [-52.337, -10.962, 81.292, 75.436, 54.875, -65.698]
  MoveL 3871 to (-26.41, 164.46, 59.84) mm, rotated rx 180 ry 0 rz 180 deg; joints [-52.337, -10.962, 81.292, 75.436, 54.875, -65.698]
  Call Extruder(396.97535)
  MoveL 3872 to (-26.72, 164.41, 59.84) mm, rotated rx 180 ry 0 rz 180 deg; joints [-52.371, -10.994, 81.318, 75.449, 54.907, -65.701]
  MoveL 3873 to (-26.72, 164.41, 59.84) mm, rotated rx 180 ry 0 rz 180 deg; joints [-52.371, -10.994, 81.318, 75.449, 54.907, -65.701]
  Call Extruder(397.13782)
  MoveL 3874 to (-27.03, 164.37, 59.84) mm, rotated rx -180 ry 0 rz 180 deg; joints [-52.405, -11.026, 81.343, 75.462, 54.94, -65.703]
  MoveL 3875 to (-27.03, 164.37, 59.84) mm, rotated rx -180 ry 0 rz 180 deg; joints [-52.405, -11.026, 81.343, 75.462, 54.94, -65.703]
  Call Extruder(397.27175)
  MoveL 3876 to (-27.28, 164.32, 59.84) mm, rotated rx 180 ry 0 rz 180 deg; joints [-52.432, -11.053, 81.365, 75.472, 54.966, -65.704]
  MoveL 3877 to (-27.28, 164.32, 59.84) mm, rotated rx 180 ry 0 rz 180 deg; joints [-52.432, -11.053, 81.365, 75.472, 54.966, -65.704]
  Call Extruder(397.40628)
  MoveL 3878 to (-27.52, 164.27, 59.84) mm, rotated rx 180 ry 0 rz 180 deg; joints [-52.459, -11.08, 81.387, 75.481, 54.992, -65.706]
  MoveL 3879 to (-27.52, 164.27, 59.84) mm, rotated rx 180 ry 0 rz 180 deg; joints [-52.459, -11.08, 81.387, 75.481, 54.992, -65.706]
  Call Extruder(397.54143)
  MoveL 3880 to (-27.77, 164.22, 59.84) mm, rotated rx 180 ry 0 rz 180 deg; joints [-52.486, -11.107, 81.409, 75.491, 55.018, -65.707]
  MoveL 3881 to (-27.77, 164.22, 59.84) mm, rotated rx 180 ry 0 rz 180 deg; joints [-52.486, -11.107, 81.409, 75.491, 55.018, -65.707]
  Call Extruder(397.67719)
  MoveL 3882 to (-28.02, 164.17, 59.84) mm, rotated rx 180 ry 0 rz 180 deg; joints [-52.513, -11.135, 81.43, 75.501, 55.044, -65.708]
  MoveL 3883 to (-28.02, 164.17, 59.84) mm, rotated rx 180 ry 0 rz 180 deg; joints [-52.513, -11.135, 81.43, 75.501, 55.044, -65.708]
  Call Extruder(397.81355)
  MoveL 3884 to (-28.27, 164.12, 59.84) mm, rotated rx 180 ry 0 rz 180 deg; joints [-52.54, -11.162, 81.452, 75.511, 55.07, -65.71]
  MoveL 3885 to (-28.27, 164.12, 59.84) mm, rotated rx 180 ry 0 rz 180 deg; joints [-52.54, -11.162, 81.452, 75.511, 55.07, -65.71]
  Call Extruder(397.89841)
  MoveL 3886 to (-28.42, 164.09, 59.84) mm, rotated rx 180 ry 0 rz -180 deg; joints [-52.556, -11.178, 81.465, 75.517, 55.086, -65.71]
  Set speed (130.0 mm/s)
  MoveL 3887 to (-31.76, 163.31, 59.84) mm, rotated rx 180 ry 0 rz 180 deg; joints [-52.91, -11.553, 81.763, 75.642, 55.427, -65.721]
  MoveL 3888 to (-31.76, 163.31, 69.25) mm, rotated rx 180 ry 0 rz 180 deg; joints [-52.91, -12.376, 83.935, 76.551, 55.103, -67.315]
  Call Extruder(395.89841)
  Set speed (40.0 mm/s)
  MoveL 3889 to (-31.76, 163.31, 69.25) mm, rotated rx 180 ry 0 rz 180 deg; joints [-52.91, -12.376, 83.935, 76.551, 55.103, -67.315]
  Call Extruder(0.00000)
  Set speed (130.0 mm/s)
  MoveL 3890 to (-31.64, 163.21, 69.25) mm, rotated rx 180 ry 0 rz 180 deg; joints [-52.884, -12.377, 83.936, 76.538, 55.079, -67.307]
  Call Extruder(2.00000)
  Set speed (40.0 mm/s)
  MoveL 3891 to (-31.64, 163.21, 69.25) mm, rotated rx 180 ry 0 rz 180 deg; joints [-52.884, -12.377, 83.936, 76.538, 55.079, -67.307]
  Set speed (30.0 mm/s)
  MoveL 3892 to (-31.64, 163.21, 69.25) mm, rotated rx 180 ry 0 rz 180 deg; joints [-52.884, -12.377, 83.936, 76.538, 55.079, -67.307]
  Call Extruder(2.18198)
  MoveL 3893 to (-31.93, 163.09, 69.25) mm, rotated rx 180 ry 0 rz 180 deg; joints [-52.91, -12.416, 83.967, 76.545, 55.105, -67.304]
  MoveL 3894 to (-31.93, 163.09, 69.25) mm, rotated rx 180 ry 0 rz 180 deg; joints [-52.91, -12.416, 83.967, 76.545, 55.105, -67.304]
  Call Extruder(2.36471)
  MoveL 3895 to (-32.22, 162.97, 69.25) mm, rotated rx -180 ry 0 rz -180 deg; joints [-52.936, -12.454, 83.997, 76.551, 55.131, -67.301]
  MoveL 3896 to (-32.22, 162.97, 69.25) mm, rotated rx -180 ry 0 rz -180 deg; joints [-52.936, -12.454, 83.997, 76.551, 55.131, -67.301]
  Call Extruder(2.53513)
  MoveL 3897 to (-32.49, 162.85, 69.25) mm, rotated rx 180 ry 0 rz 180 deg; joints [-52.96, -12.49, 84.025, 76.557, 55.155, -67.298]
  MoveL 3898 to (-32.49, 162.85, 69.25) mm, rotated rx 180 ry 0 rz 180 deg; joints [-52.96, -12.49, 84.025, 76.557, 55.155, -67.298]
  Call Extruder(2.69310)
  MoveL 3899 to (-32.74, 162.74, 69.25) mm, rotated rx -180 ry 0 rz 180 deg; joints [-52.982, -12.524, 84.051, 76.562, 55.177, -67.295]
  MoveL 3900 to (-32.74, 162.74, 69.25) mm, rotated rx -180 ry 0 rz 180 deg; joints [-52.982, -12.524, 84.051, 76.562, 55.177, -67.295]
  Call Extruder(2.85168)
  MoveL 3901 to (-32.99, 162.64, 69.25) mm, rotated rx -180 ry 0 rz -180 deg; joints [-53.004, -12.557, 84.077, 76.568, 55.199, -67.292]
  MoveL 3902 to (-32.99, 162.64, 69.25) mm, rotated rx -180 ry 0 rz -180 deg; joints [-53.004, -12.557, 84.077, 76.568, 55.199, -67.292]
  Call Extruder(3.05784)
  MoveL 3903 to (-33.29, 162.46, 69.25) mm, rotated rx 180 ry 0 rz 180 deg; joints [-53.026, -12.603, 84.112, 76.571, 55.222, -67.286]
  MoveL 3904 to (-33.29, 162.46, 69.25) mm, rotated rx 180 ry 0 rz 180 deg; joints [-53.026, -12.603, 84.112, 76.571, 55.222, -67.286]
  Call Extruder(3.26479)
  MoveL 3905 to (-33.6, 162.29, 69.25) mm, rotated rx 180 ry 0 rz 180 deg; joints [-53.049, -12.649, 84.148, 76.575, 55.245, -67.28]
  MoveL 3906 to (-33.6, 162.29, 69.25) mm, rotated rx 180 ry 0 rz 180 deg; joints [-53.049, -12.649, 84.148, 76.575, 55.245, -67.28]
  Call Extruder(3.47251)
  MoveL 3907 to (-33.9, 162.11, 69.25) mm, rotated rx -180 ry 0 rz 180 deg; joints [-53.071, -12.695, 84.183, 76.579, 55.268, -67.274]
  MoveL 3908 to (-33.9, 162.11, 69.25) mm, rotated rx -180 ry 0 rz 180 deg; joints [-53.071, -12.695, 84.183, 76.579, 55.268, -67.274]
  Call Extruder(3.68101)
  MoveL 3909 to (-34.21, 161.94, 69.25) mm, rotated rx 180 ry 0 rz 180 deg; joints [-53.094, -12.74, 84.219, 76.582, 55.291, -67.268]
  MoveL 3910 to (-34.21, 161.94, 69.25) mm, rotated rx 180 ry 0 rz 180 deg; joints [-53.094, -12.74, 84.219, 76.582, 55.291, -67.268]
  Call Extruder(3.86055)
  MoveL 3911 to (-34.45, 161.76, 69.25) mm, rotated rx 180 ry 0 rz 180 deg; joints [-53.109, -12.781, 84.25, 76.583, 55.307, -67.261]
  MoveL 3912 to (-34.45, 161.76, 69.25) mm, rotated rx 180 ry 0 rz 180 deg; joints [-53.109, -12.781, 84.25, 76.583, 55.307, -67.261]
  Call Extruder(4.19399)
  MoveL 3913 to (-34.9, 161.43, 69.25) mm, rotated rx 180 ry 0 rz 180 deg; joints [-53.135, -12.857, 84.308, 76.584, 55.336, -67.248]
  MoveL 3914 to (-34.9, 161.43, 69.25) mm, rotated rx 180 ry 0 rz 180 deg; joints [-53.135, -12.857, 84.308, 76.584, 55.336, -67.248]
  Call Extruder(4.52861)
  MoveL 3915 to (-35.35, 161.1, 69.25) mm, rotated rx -180 ry 0 rz -180 deg; joints [-53.163, -12.932, 84.367, 76.585, 55.365, -67.234]
  Call Extruder(5.35652)
  MoveL 3916 to (-36.39, 160.19, 69.25) mm, rotated rx -180 ry 0 rz 180 deg; joints [-53.209, -13.123, 84.513, 76.577, 55.418, -67.195]
  Call Extruder(5.98652)
  MoveL 3917 to (-37.09, 159.41, 69.25) mm, rotated rx 180 ry 0 rz -180 deg; joints [-53.224, -13.271, 84.627, 76.561, 55.44, -67.157]
  Call Extruder(6.31951)
  MoveL 3918 to (-37.44, 158.97, 69.25) mm, rotated rx 180 ry 0 rz 180 deg; joints [-53.227, -13.349, 84.686, 76.55, 55.447, -67.136]
  MoveL 3919 to (-37.44, 158.97, 69.25) mm, rotated rx 180 ry 0 rz 180 deg; joints [-53.227, -13.349, 84.686, 76.55, 55.447, -67.136]
  Call Extruder(6.58931)
  MoveL 3920 to (-37.7, 158.61, 69.25) mm, rotated rx 180 ry 0 rz -180 deg; joints [-53.226, -13.413, 84.735, 76.539, 55.45, -67.118]
  Set speed (130.0 mm/s)
  MoveL 3921 to (-37.7, 158.61, 69.25) mm, rotated rx 180 ry 0 rz -180 deg; joints [-53.226, -13.413, 84.735, 76.539, 55.45, -67.118]
  Set speed (30.0 mm/s)
  MoveL 3922 to (-37.7, 158.61, 69.25) mm, rotated rx 180 ry 0 rz -180 deg; joints [-53.226, -13.413, 84.735, 76.539, 55.45, -67.118]
  Call Extruder(6.87472)
  MoveL 3923 to (-37.98, 158.22, 69.25) mm, rotated rx 180 ry 0 rz 180 deg; joints [-53.225, -13.481, 84.786, 76.528, 55.452, -67.099]
  MoveL 3924 to (-37.98, 158.22, 69.25) mm, rotated rx 180 ry 0 rz 180 deg; joints [-53.225, -13.481, 84.786, 76.528, 55.452, -67.099]
  Call Extruder(7.13432)
  MoveL 3925 to (-38.22, 157.85, 69.25) mm, rotated rx 180 ry 0 rz 180 deg; joints [-53.221, -13.542, 84.833, 76.516, 55.452, -67.08]
  MoveL 3926 to (-38.22, 157.85, 69.25) mm, rotated rx 180 ry 0 rz 180 deg; joints [-53.221, -13.542, 84.833, 76.516, 55.452, -67.08]
  Call Extruder(7.34204)
  MoveL 3927 to (-38.4, 157.55, 69.25) mm, rotated rx 180 ry 0 rz 180 deg; joints [-53.214, -13.591, 84.87, 76.505, 55.448, -67.064]
  MoveL 3928 to (-38.4, 157.55, 69.25) mm, rotated rx 180 ry 0 rz 180 deg; joints [-53.214, -13.591, 84.87, 76.505, 55.448, -67.064]
  Call Extruder(7.54898)
  MoveL 3929 to (-38.57, 157.25, 69.25) mm, rotated rx 180 ry 0 rz 180 deg; joints [-53.207, -13.64, 84.907, 76.494, 55.445, -67.048]
  MoveL 3930 to (-38.57, 157.25, 69.25) mm, rotated rx 180 ry 0 rz 180 deg; joints [-53.207, -13.64, 84.907, 76.494, 55.445, -67.048]
  Call Extruder(7.75514)
  MoveL 3931 to (-38.75, 156.94, 69.25) mm, rotated rx 180 ry 0 rz 180 deg; joints [-53.2, -13.689, 84.944, 76.482, 55.441, -67.033]
  MoveL 3932 to (-38.75, 156.94, 69.25) mm, rotated rx 180 ry 0 rz 180 deg; joints [-53.2, -13.689, 84.944, 76.482, 55.441, -67.033]
  Call Extruder(7.93681)
  MoveL 3933 to (-38.89, 156.66, 69.25) mm, rotated rx 180 ry 0 rz 180 deg; joints [-53.191, -13.732, 84.977, 76.471, 55.435, -67.018]
  MoveL 3934 to (-38.89, 156.66, 69.25) mm, rotated rx 180 ry 0 rz 180 deg; joints [-53.191, -13.732, 84.977, 76.471, 55.435, -67.018]
  Call Extruder(8.09480)
  MoveL 3935 to (-39, 156.42, 69.25) mm, rotated rx 180 ry 0 rz 180 deg; joints [-53.18, -13.769, 85.005, 76.46, 55.428, -67.004]
  MoveL 3936 to (-39, 156.42, 69.25) mm, rotated rx 180 ry 0 rz 180 deg; joints [-53.18, -13.769, 85.005, 76.46, 55.428, -67.004]
  Call Extruder(8.25218)
  MoveL 3937 to (-39.1, 156.17, 69.25) mm, rotated rx -180 ry 0 rz -180 deg; joints [-53.17, -13.807, 85.033, 76.449, 55.42, -66.991]
  MoveL 3938 to (-39.1, 156.17, 69.25) mm, rotated rx -180 ry 0 rz -180 deg; joints [-53.17, -13.807, 85.033, 76.449, 55.42, -66.991]
  Call Extruder(8.43490)
  MoveL 3939 to (-39.23, 155.87, 69.25) mm, rotated rx 180 ry 0 rz 180 deg; joints [-53.156, -13.849, 85.065, 76.435, 55.41, -66.975]
  MoveL 3940 to (-39.23, 155.87, 69.25) mm, rotated rx 180 ry 0 rz 180 deg; joints [-53.156, -13.849, 85.065, 76.435, 55.41, -66.975]
  Call Extruder(8.61686)
  MoveL 3941 to (-39.35, 155.58, 69.25) mm, rotated rx 180 ry 0 rz 180 deg; joints [-53.143, -13.893, 85.098, 76.422, 55.401, -66.958]
  MoveL 3942 to (-39.35, 155.58, 69.25) mm, rotated rx 180 ry 0 rz 180 deg; joints [-53.143, -13.893, 85.098, 76.422, 55.401, -66.958]
  Call Extruder(8.76420)
  MoveL 3943 to (-39.44, 155.34, 69.25) mm, rotated rx 180 ry 0 rz 180 deg; joints [-53.131, -13.927, 85.124, 76.411, 55.392, -66.945]
  MoveL 3944 to (-39.44, 155.34, 69.25) mm, rotated rx 180 ry 0 rz 180 deg; joints [-53.131, -13.927, 85.124, 76.411, 55.392, -66.945]
  Call Extruder(8.87743)
  MoveL 3945 to (-39.5, 155.15, 69.25) mm, rotated rx 180 ry 0 rz 180 deg; joints [-53.121, -13.954, 85.144, 76.401, 55.384, -66.934]
  MoveL 3946 to (-39.5, 155.15, 69.25) mm, rotated rx 180 ry 0 rz 180 deg; joints [-53.121, -13.954, 85.144, 76.401, 55.384, -66.934]
  Call Extruder(8.99022)
  MoveL 3947 to (-39.56, 154.97, 69.25) mm, rotated rx 180 ry 0 rz 180 deg; joints [-53.11, -13.98, 85.164, 76.392, 55.375, -66.924]
  MoveL 3948 to (-39.56, 154.97, 69.25) mm, rotated rx 180 ry 0 rz 180 deg; joints [-53.11, -13.98, 85.164, 76.392, 55.375, -66.924]
  Call Extruder(9.10257)
  MoveL 3949 to (-39.62, 154.78, 69.25) mm, rotated rx 180 ry 0 rz 180 deg; joints [-53.099, -14.006, 85.183, 76.382, 55.367, -66.913]
  MoveL 3950 to (-39.62, 154.78, 69.25) mm, rotated rx 180 ry 0 rz 180 deg; joints [-53.099, -14.006, 85.183, 76.382, 55.367, -66.913]
  Call Extruder(9.21447)
  MoveL 3951 to (-39.68, 154.59, 69.25) mm, rotated rx 180 ry 0 rz 180 deg; joints [-53.088, -14.033, 85.203, 76.373, 55.358, -66.902]
  MoveL 3952 to (-39.68, 154.59, 69.25) mm, rotated rx 180 ry 0 rz 180 deg; joints [-53.088, -14.033, 85.203, 76.373, 55.358, -66.902]
  Call Extruder(9.33587)
  MoveL 3953 to (-39.75, 154.38, 69.25) mm, rotated rx 180 ry 0 rz -180 deg; joints [-53.076, -14.061, 85.225, 76.362, 55.349, -66.891]
  MoveL 3954 to (-39.75, 154.38, 69.25) mm, rotated rx 180 ry 0 rz -180 deg; joints [-53.076, -14.061, 85.225, 76.362, 55.349, -66.891]
  Call Extruder(9.46666)
  MoveL 3955 to (-39.81, 154.16, 69.25) mm, rotated rx 180 ry 0 rz 180 deg; joints [-53.063, -14.092, 85.248, 76.35, 55.338, -66.878]
  MoveL 3956 to (-39.81, 154.16, 69.25) mm, rotated rx 180 ry 0 rz 180 deg; joints [-53.063, -14.092, 85.248, 76.35, 55.338, -66.878]
  Call Extruder(9.59689)
  MoveL 3957 to (-39.88, 153.94, 69.25) mm, rotated rx 180 ry 0 rz 180 deg; joints [-53.049, -14.123, 85.271, 76.339, 55.328, -66.865]
  MoveL 3958 to (-39.88, 153.94, 69.25) mm, rotated rx 180 ry 0 rz 180 deg; joints [-53.049, -14.123, 85.271, 76.339, 55.328, -66.865]
  Call Extruder(9.72656)
  MoveL 3959 to (-39.95, 153.71, 69.25) mm, rotated rx 180 ry 0 rz 180 deg; joints [-53.036, -14.154, 85.294, 76.327, 55.317, -66.852]
  MoveL 3960 to (-39.95, 153.71, 69.25) mm, rotated rx 180 ry 0 rz 180 deg; joints [-53.036, -14.154, 85.294, 76.327, 55.317, -66.852]
  Call Extruder(9.85565)
  MoveL 3961 to (-40.02, 153.49, 69.25) mm, rotated rx 180 ry 0 rz 180 deg; joints [-53.022, -14.184, 85.317, 76.315, 55.306, -66.839]
  MoveL 3962 to (-40.02, 153.49, 69.25) mm, rotated rx 180 ry 0 rz 180 deg; joints [-53.022, -14.184, 85.317, 76.315, 55.306, -66.839]
  Call Extruder(9.97074)
  MoveL 3963 to (-40.06, 153.28, 69.25) mm, rotated rx 180 ry 0 rz 180 deg; joints [-53.007, -14.211, 85.337, 76.304, 55.294, -66.827]
  MoveL 3964 to (-40.06, 153.28, 69.25) mm, rotated rx 180 ry 0 rz 180 deg; joints [-53.007, -14.211, 85.337, 76.304, 55.294, -66.827]
  Call Extruder(10.08538)
  MoveL 3965 to (-40.11, 153.08, 69.25) mm, rotated rx 180 ry 0 rz 180 deg; joints [-52.993, -14.238, 85.357, 76.292, 55.283, -66.815]
  MoveL 3966 to (-40.11, 153.08, 69.25) mm, rotated rx 180 ry 0 rz 180 deg; joints [-52.993, -14.238, 85.357, 76.292, 55.283, -66.815]
  Call Extruder(10.19956)
  MoveL 3967 to (-40.15, 152.88, 69.25) mm, rotated rx 180 ry 0 rz -180 deg; joints [-52.978, -14.264, 85.376, 76.281, 55.271, -66.803]
  MoveL 3968 to (-40.15, 152.88, 69.25) mm, rotated rx 180 ry 0 rz -180 deg; joints [-52.978, -14.264, 85.376, 76.281, 55.271, -66.803]
  Call Extruder(10.31329)
  MoveL 3969 to (-40.2, 152.67, 69.25) mm, rotated rx 180 ry 0 rz 180 deg; joints [-52.963, -14.291, 85.396, 76.269, 55.259, -66.791]
  MoveL 3970 to (-40.2, 152.67, 69.25) mm, rotated rx 180 ry 0 rz 180 deg; joints [-52.963, -14.291, 85.396, 76.269, 55.259, -66.791]
  Call Extruder(10.43872)
  MoveL 3971 to (-40.24, 152.44, 69.25) mm, rotated rx -180 ry 0 rz 180 deg; joints [-52.946, -14.32, 85.418, 76.256, 55.245, -66.778]
  MoveL 3972 to (-40.24, 152.44, 69.25) mm, rotated rx -180 ry 0 rz 180 deg; joints [-52.946, -14.32, 85.418, 76.256, 55.245, -66.778]
  Call Extruder(10.57569)
  MoveL 3973 to (-40.29, 152.2, 69.25) mm, rotated rx 180 ry 0 rz 180 deg; joints [-52.928, -14.352, 85.442, 76.241, 55.23, -66.763]
  MoveL 3974 to (-40.29, 152.2, 69.25) mm, rotated rx 180 ry 0 rz 180 deg; joints [-52.928, -14.352, 85.442, 76.241, 55.23, -66.763]
  Call Extruder(10.71206)
  MoveL 3975 to (-40.34, 151.95, 69.25) mm, rotated rx 180 ry 0 rz 180 deg; joints [-52.909, -14.384, 85.466, 76.227, 55.214, -66.748]
  MoveL 3976 to (-40.34, 151.95, 69.25) mm, rotated rx 180 ry 0 rz 180 deg; joints [-52.909, -14.384, 85.466, 76.227, 55.214, -66.748]
  Call Extruder(10.84781)
  MoveL 3977 to (-40.39, 151.7, 69.25) mm, rotated rx 180 ry 0 rz 180 deg; joints [-52.89, -14.416, 85.49, 76.212, 55.199, -66.733]
  MoveL 3978 to (-40.39, 151.7, 69.25) mm, rotated rx 180 ry 0 rz 180 deg; joints [-52.89, -14.416, 85.49, 76.212, 55.199, -66.733]
  Call Extruder(10.98296)
  MoveL 3979 to (-40.44, 151.45, 69.25) mm, rotated rx -180 ry 0 rz 180 deg; joints [-52.871, -14.448, 85.513, 76.198, 55.184, -66.719]
  MoveL 3980 to (-40.44, 151.45, 69.25) mm, rotated rx -180 ry 0 rz 180 deg; joints [-52.871, -14.448, 85.513, 76.198, 55.184, -66.719]
  Call Extruder(11.11749)
  MoveL 3981 to (-40.49, 151.2, 69.25) mm, rotated rx 180 ry 0 rz 180 deg; joints [-52.853, -14.48, 85.537, 76.183, 55.169, -66.704]
  MoveL 3982 to (-40.49, 151.2, 69.25) mm, rotated rx 180 ry 0 rz 180 deg; joints [-52.853, -14.48, 85.537, 76.183, 55.169, -66.704]
  Call Extruder(11.25142)
  MoveL 3983 to (-40.54, 150.95, 69.25) mm, rotated rx 180 ry 0 rz 180 deg; joints [-52.834, -14.512, 85.561, 76.168, 55.153, -66.689]
  MoveL 3984 to (-40.54, 150.95, 69.25) mm, rotated rx 180 ry 0 rz 180 deg; joints [-52.834, -14.512, 85.561, 76.168, 55.153, -66.689]
  Call Extruder(11.39927)
  MoveL 3985 to (-40.59, 150.67, 69.25) mm, rotated rx 180 ry 0 rz 180 deg; joints [-52.812, -14.547, 85.587, 76.152, 55.135, -66.672]
  MoveL 3986 to (-40.59, 150.67, 69.25) mm, rotated rx 180 ry 0 rz 180 deg; joints [-52.812, -14.547, 85.587, 76.152, 55.135, -66.672]
  Call Extruder(11.56100)
  MoveL 3987 to (-40.64, 150.37, 69.25) mm, rotated rx 180 ry 0 rz 180 deg; joints [-52.787, -14.586, 85.615, 76.133, 55.115, -66.653]
  MoveL 3988 to (-40.64, 150.37, 69.25) mm, rotated rx 180 ry 0 rz 180 deg; joints [-52.787, -14.586, 85.615, 76.133, 55.115, -66.653]
  Call Extruder(11.72199)
  MoveL 3989 to (-40.69, 150.06, 69.25) mm, rotated rx 180 ry 0 rz 180 deg; joints [-52.762, -14.624, 85.643, 76.114, 55.094, -66.635]
  MoveL 3990 to (-40.69, 150.06, 69.25) mm, rotated rx 180 ry 0 rz 180 deg; joints [-52.762, -14.624, 85.643, 76.114, 55.094, -66.635]
  Call Extruder(11.88226)
  MoveL 3991 to (-40.74, 149.76, 69.25) mm, rotated rx 180 ry 0 rz 180 deg; joints [-52.737, -14.662, 85.672, 76.095, 55.074, -66.616]
  MoveL 3992 to (-40.74, 149.76, 69.25) mm, rotated rx 180 ry 0 rz 180 deg; joints [-52.737, -14.662, 85.672, 76.095, 55.074, -66.616]
  Call Extruder(12.04180)
  MoveL 3993 to (-40.78, 149.45, 69.25) mm, rotated rx 180 ry 0 rz 180 deg; joints [-52.712, -14.7, 85.7, 76.077, 55.053, -66.597]
  MoveL 3994 to (-40.78, 149.45, 69.25) mm, rotated rx 180 ry 0 rz 180 deg; joints [-52.712, -14.7, 85.7, 76.077, 55.053, -66.597]
  Call Extruder(12.20062)
  MoveL 3995 to (-40.83, 149.14, 69.25) mm, rotated rx -180 ry 0 rz -180 deg; joints [-52.687, -14.738, 85.728, 76.058, 55.033, -66.579]
  MoveL 3996 to (-40.83, 149.14, 69.25) mm, rotated rx -180 ry 0 rz -180 deg; joints [-52.687, -14.738, 85.728, 76.058, 55.033, -66.579]
  Call Extruder(12.37928)
  MoveL 3997 to (-40.88, 148.8, 69.25) mm, rotated rx 180 ry 0 rz 180 deg; joints [-52.658, -14.78, 85.759, 76.036, 55.009, -66.557]
  MoveL 3998 to (-40.88, 148.8, 69.25) mm, rotated rx 180 ry 0 rz 180 deg; joints [-52.658, -14.78, 85.759, 76.036, 55.009, -66.557]
  Call Extruder(12.57772)
  MoveL 3999 to (-40.92, 148.41, 69.25) mm, rotated rx -180 ry 0 rz 180 deg; joints [-52.624, -14.827, 85.794, 76.011, 54.98, -66.533]
  MoveL 4000 to (-40.92, 148.41, 69.25) mm, rotated rx -180 ry 0 rz 180 deg; joints [-52.624, -14.827, 85.794, 76.011, 54.98, -66.533]
  Call Extruder(12.77530)
  MoveL 4001 to (-40.97, 148.02, 69.25) mm, rotated rx -180 ry 0 rz 180 deg; joints [-52.59, -14.874, 85.828, 75.986, 54.952, -66.509]
  MoveL 4002 to (-40.97, 148.02, 69.25) mm, rotated rx -180 ry 0 rz 180 deg; joints [-52.59, -14.874, 85.828, 75.986, 54.952, -66.509]
  Call Extruder(12.97200)
  MoveL 4003 to (-41.02, 147.63, 69.25) mm, rotated rx -180 ry 0 rz 180 deg; joints [-52.556, -14.921, 85.863, 75.961, 54.924, -66.484]
  MoveL 4004 to (-41.02, 147.63, 69.25) mm, rotated rx -180 ry 0 rz 180 deg; joints [-52.556, -14.921, 85.863, 75.961, 54.924, -66.484]
  Call Extruder(13.16784)
  MoveL 4005 to (-41.06, 147.25, 69.25) mm, rotated rx 180 ry 0 rz -180 deg; joints [-52.521, -14.968, 85.897, 75.936, 54.896, -66.46]
  MoveL 4006 to (-41.06, 147.25, 69.25) mm, rotated rx 180 ry 0 rz -180 deg; joints [-52.521, -14.968, 85.897, 75.936, 54.896, -66.46]
  Call Extruder(13.46324)
  MoveL 4007 to (-41.11, 146.66, 69.25) mm, rotated rx -180 ry 0 rz 180 deg; joints [-52.466, -15.037, 85.948, 75.896, 54.849, -66.423]
  MoveL 4008 to (-41.11, 146.66, 69.25) mm, rotated rx -180 ry 0 rz 180 deg; joints [-52.466, -15.037, 85.948, 75.896, 54.849, -66.423]
  Call Extruder(13.75731)
  MoveL 4009 to (-41.15, 146.07, 69.25) mm, rotated rx 180 ry 0 rz 180 deg; joints [-52.411, -15.106, 85.998, 75.856, 54.803, -66.385]
  MoveL 4010 to (-41.15, 146.07, 69.25) mm, rotated rx 180 ry 0 rz 180 deg; joints [-52.411, -15.106, 85.998, 75.856, 54.803, -66.385]
  Call Extruder(14.05004)
  MoveL 4011 to (-41.2, 145.48, 69.25) mm, rotated rx 180 ry 0 rz -180 deg; joints [-52.355, -15.175, 86.049, 75.816, 54.757, -66.347]
  MoveL 4012 to (-41.2, 145.48, 69.25) mm, rotated rx 180 ry 0 rz -180 deg; joints [-52.355, -15.175, 86.049, 75.816, 54.757, -66.347]
  Call Extruder(14.62350)
  MoveL 4013 to (-41.25, 144.32, 69.25) mm, rotated rx 180 ry 0 rz 180 deg; joints [-52.239, -15.307, 86.145, 75.734, 54.659, -66.271]
  MoveL 4014 to (-41.25, 144.32, 69.25) mm, rotated rx 180 ry 0 rz 180 deg; joints [-52.239, -15.307, 86.145, 75.734, 54.659, -66.271]
  Call Extruder(15.33745)
  MoveL 4015 to (-41.29, 142.86, 69.25) mm, rotated rx 180 ry 0 rz -180 deg; joints [-52.09, -15.471, 86.263, 75.63, 54.534, -66.175]
  Call Extruder(57.40228)
  MoveL 4016 to (-41.29, 57.14, 69.25) mm, rotated rx -180 ry 0 rz -180 deg; joints [-40.759, -23.907, 91.713, 66.334, 45.465, -57.999]
  Call Extruder(57.83083)
  MoveL 4017 to (-41.27, 56.26, 69.25) mm, rotated rx 180 ry 0 rz -180 deg; joints [-40.614, -23.98, 91.754, 66.197, 45.356, -57.882]
  MoveL 4018 to (-41.27, 56.26, 69.25) mm, rotated rx 180 ry 0 rz -180 deg; joints [-40.614, -23.98, 91.754, 66.197, 45.356, -57.882]
  Call Extruder(58.40429)
  MoveL 4019 to (-41.22, 55.1, 69.25) mm, rotated rx -180 ry 0 rz 180 deg; joints [-40.419, -24.075, 91.807, 66.013, 45.207, -57.726]
  MoveL 4020 to (-41.22, 55.1, 69.25) mm, rotated rx -180 ry 0 rz 180 deg; joints [-40.419, -24.075, 91.807, 66.013, 45.207, -57.726]
  Call Extruder(58.83860)
  MoveL 4021 to (-41.18, 54.23, 69.25) mm, rotated rx 180 ry 0 rz 180 deg; joints [-40.269, -24.145, 91.846, 65.872, 45.093, -57.607]
  MoveL 4022 to (-41.18, 54.23, 69.25) mm, rotated rx 180 ry 0 rz 180 deg; joints [-40.269, -24.145, 91.846, 65.872, 45.093, -57.607]
  Call Extruder(59.13267)
  MoveL 4023 to (-41.13, 53.64, 69.25) mm, rotated rx 180 ry 0 rz 180 deg; joints [-40.165, -24.19, 91.872, 65.776, 45.013, -57.526]
  MoveL 4024 to (-41.13, 53.64, 69.25) mm, rotated rx 180 ry 0 rz 180 deg; joints [-40.165, -24.19, 91.872, 65.776, 45.013, -57.526]
  Call Extruder(59.42806)
  MoveL 4025 to (-41.09, 53.05, 69.25) mm, rotated rx 180 ry 0 rz -180 deg; joints [-40.062, -24.235, 91.897, 65.679, 44.934, -57.445]
  MoveL 4026 to (-41.09, 53.05, 69.25) mm, rotated rx 180 ry 0 rz -180 deg; joints [-40.062, -24.235, 91.897, 65.679, 44.934, -57.445]
  Call Extruder(59.67430)
  MoveL 4027 to (-41.04, 52.56, 69.25) mm, rotated rx -180 ry 0 rz 180 deg; joints [-39.975, -24.271, 91.918, 65.598, 44.867, -57.377]
  MoveL 4028 to (-41.04, 52.56, 69.25) mm, rotated rx -180 ry 0 rz 180 deg; joints [-39.975, -24.271, 91.918, 65.598, 44.867, -57.377]
  Call Extruder(59.87100)
  MoveL 4029 to (-40.99, 52.17, 69.25) mm, rotated rx -180 ry 0 rz 180 deg; joints [-39.904, -24.299, 91.933, 65.533, 44.813, -57.323]
  MoveL 4030 to (-40.99, 52.17, 69.25) mm, rotated rx -180 ry 0 rz 180 deg; joints [-39.904, -24.299, 91.933, 65.533, 44.813, -57.323]
  Call Extruder(60.06858)
  MoveL 4031 to (-40.95, 51.78, 69.25) mm, rotated rx -180 ry 0 rz 180 deg; joints [-39.833, -24.327, 91.949, 65.467, 44.759, -57.268]
  MoveL 4032 to (-40.95, 51.78, 69.25) mm, rotated rx -180 ry 0 rz 180 deg; joints [-39.833, -24.327, 91.949, 65.467, 44.759, -57.268]
  Call Extruder(60.26702)
  MoveL 4033 to (-40.9, 51.4, 69.25) mm, rotated rx 180 ry 0 rz 180 deg; joints [-39.763, -24.355, 91.964, 65.401, 44.704, -57.214]
  MoveL 4034 to (-40.9, 51.4, 69.25) mm, rotated rx 180 ry 0 rz 180 deg; joints [-39.763, -24.355, 91.964, 65.401, 44.704, -57.214]
  Call Extruder(60.46633)
  MoveL 4035 to (-40.86, 51.01, 69.25) mm, rotated rx 180 ry 0 rz 180 deg; joints [-39.692, -24.383, 91.98, 65.335, 44.65, -57.159]
  MoveL 4036 to (-40.86, 51.01, 69.25) mm, rotated rx 180 ry 0 rz 180 deg; joints [-39.692, -24.383, 91.98, 65.335, 44.65, -57.159]
  Call Extruder(60.62514)
  MoveL 4037 to (-40.81, 50.7, 69.25) mm, rotated rx -180 ry 0 rz 180 deg; joints [-39.634, -24.404, 91.991, 65.282, 44.605, -57.115]
  MoveL 4038 to (-40.81, 50.7, 69.25) mm, rotated rx -180 ry 0 rz 180 deg; joints [-39.634, -24.404, 91.991, 65.282, 44.605, -57.115]
  Call Extruder(60.78469)
  MoveL 4039 to (-40.76, 50.4, 69.25) mm, rotated rx -180 ry 0 rz 180 deg; joints [-39.576, -24.424, 92.003, 65.229, 44.56, -57.072]
  MoveL 4040 to (-40.76, 50.4, 69.25) mm, rotated rx -180 ry 0 rz 180 deg; joints [-39.576, -24.424, 92.003, 65.229, 44.56, -57.072]
  Call Extruder(60.94496)
  MoveL 4041 to (-40.71, 50.09, 69.25) mm, rotated rx 180 ry 0 rz 180 deg; joints [-39.518, -24.445, 92.014, 65.176, 44.516, -57.028]
  MoveL 4042 to (-40.71, 50.09, 69.25) mm, rotated rx 180 ry 0 rz 180 deg; joints [-39.518, -24.445, 92.014, 65.176, 44.516, -57.028]
  Call Extruder(61.10596)
  MoveL 4043 to (-40.66, 49.79, 69.25) mm, rotated rx 180 ry 0 rz 180 deg; joints [-39.46, -24.465, 92.026, 65.123, 44.471, -56.984]
  MoveL 4044 to (-40.66, 49.79, 69.25) mm, rotated rx 180 ry 0 rz 180 deg; joints [-39.46, -24.465, 92.026, 65.123, 44.471, -56.984]
  Call Extruder(61.26769)
  MoveL 4045 to (-40.61, 49.48, 69.25) mm, rotated rx 180 ry 0 rz 180 deg; joints [-39.402, -24.486, 92.037, 65.069, 44.426, -56.94]
  MoveL 4046 to (-40.61, 49.48, 69.25) mm, rotated rx 180 ry 0 rz 180 deg; joints [-39.402, -24.486, 92.037, 65.069, 44.426, -56.94]
  Call Extruder(61.43014)
  MoveL 4047 to (-40.56, 49.17, 69.25) mm, rotated rx 180 ry 0 rz 180 deg; joints [-39.344, -24.506, 92.048, 65.015, 44.382, -56.896]
  MoveL 4048 to (-40.56, 49.17, 69.25) mm, rotated rx 180 ry 0 rz 180 deg; joints [-39.344, -24.506, 92.048, 65.015, 44.382, -56.896]
  Call Extruder(61.56407)
  MoveL 4049 to (-40.52, 48.93, 69.25) mm, rotated rx 180 ry 0 rz 180 deg; joints [-39.296, -24.522, 92.057, 64.971, 44.344, -56.859]
  MoveL 4050 to (-40.52, 48.93, 69.25) mm, rotated rx 180 ry 0 rz 180 deg; joints [-39.296, -24.522, 92.057, 64.971, 44.344, -56.859]
  Call Extruder(61.69860)
  MoveL 4051 to (-40.47, 48.68, 69.25) mm, rotated rx -180 ry 0 rz 180 deg; joints [-39.247, -24.538, 92.066, 64.926, 44.306, -56.823]
  MoveL 4052 to (-40.47, 48.68, 69.25) mm, rotated rx -180 ry 0 rz 180 deg; joints [-39.247, -24.538, 92.066, 64.926, 44.306, -56.823]
  Call Extruder(61.83375)
  MoveL 4053 to (-40.42, 48.43, 69.25) mm, rotated rx 180 ry 0 rz 180 deg; joints [-39.198, -24.553, 92.074, 64.881, 44.268, -56.787]
  MoveL 4054 to (-40.42, 48.43, 69.25) mm, rotated rx 180 ry 0 rz 180 deg; joints [-39.198, -24.553, 92.074, 64.881, 44.268, -56.787]
  Call Extruder(61.96950)
  MoveL 4055 to (-40.37, 48.18, 69.25) mm, rotated rx 180 ry 0 rz 180 deg; joints [-39.149, -24.569, 92.083, 64.836, 44.23, -56.75]
  MoveL 4056 to (-40.37, 48.18, 69.25) mm, rotated rx 180 ry 0 rz 180 deg; joints [-39.149, -24.569, 92.083, 64.836, 44.23, -56.75]
  Call Extruder(62.10587)
  MoveL 4057 to (-40.32, 47.93, 69.25) mm, rotated rx 180 ry 0 rz 180 deg; joints [-39.1, -24.584, 92.091, 64.792, 44.192, -56.714]
  MoveL 4058 to (-40.32, 47.93, 69.25) mm, rotated rx 180 ry 0 rz 180 deg; joints [-39.1, -24.584, 92.091, 64.792, 44.192, -56.714]
  Call Extruder(62.24285)
  MoveL 4059 to (-40.27, 47.68, 69.25) mm, rotated rx -180 ry 0 rz 180 deg; joints [-39.051, -24.6, 92.1, 64.747, 44.154, -56.677]
  MoveL 4060 to (-40.27, 47.68, 69.25) mm, rotated rx -180 ry 0 rz 180 deg; joints [-39.051, -24.6, 92.1, 64.747, 44.154, -56.677]
  Call Extruder(62.38043)
  MoveL 4061 to (-40.22, 47.43, 69.25) mm, rotated rx 180 ry 0 rz -180 deg; joints [-39.002, -24.615, 92.109, 64.701, 44.116, -56.64]
